LIN {X 0,Y 504.694,Z 139.15,A -85,B 0,C 180,E1 19601.04,E2 19601.04} C_VEL
LIN {X 0,Y 504.678,Z 139.182,A -85,B 0,C 180,E1 19597.642,E2 19597.642} C_VEL
LIN {X 0,Y 504.643,Z 139.158,A -85,B 0,C 180,E1 19594.284,E2 19594.284} C_VEL
LIN {X 0,Y 504.674,Z 139.176,A -85,B 0,C 180,E1 19590.889,E2 19590.889} C_VEL
LIN {X 0,Y 504.678,Z 139.173,A -85,B 0,C 180,E1 19587.527,E2 19587.527} C_VEL
LIN {X 0,Y 504.634,Z 139.159,A -85,B 0,C 180,E1 19584.13,E2 19584.13} C_VEL
LIN {X 0,Y 504.641,Z 139.168,A -85,B 0,C 180,E1 19580.597,E2 19580.597} C_VEL
LIN {X 0,Y 504.688,Z 139.169,A -85,B 0,C 180,E1 19577.193,E2 19577.193} C_VEL
LIN {X 0,Y 504.672,Z 139.48,A -85,B 0,C 180,E1 19576.287,E2 19576.287} C_VEL
LIN {X 0,Y 506.039,Z 142.777,A -85,B 0,C 180,E1 19575.775,E2 19575.775} C_VEL
LIN {X 0,Y 507.07,Z 144.526,A -85,B 0,C 180,E1 19575.494,E2 19575.494} C_VEL
LIN {X 0,Y 515.267,Z 161.516,A -85,B 0,C 180,E1 19573.08,E2 19573.08} C_VEL
LIN {X 0,Y 516.742,Z 164.473,A -85,B 0,C 180,E1 19572.673,E2 19572.673} C_VEL
LIN {X 0,Y 517.647,Z 168.38,A -85,B 0,C 180,E1 19572.251,E2 19572.251} C_VEL
LIN {X 0,Y 517.411,Z 174.74,A -85,B 0,C 180,E1 19571.749,E2 19571.749} C_VEL
LIN {X 0,Y 513.948,Z 193.541,A -85,B 0,C 180,E1 19570.561,E2 19570.561} C_VEL
LIN {X 0,Y 513.871,Z 194.507,A -85,B 0,C 180,E1 19570.49,E2 19570.49} C_VEL
LIN {X 0,Y 513.152,Z 207.74,A -85,B 0,C 180,E1 19569.537,E2 19569.537} C_VEL
LIN {X 0,Y 516.89,Z 230.706,A -85,B 0,C 180,E1 19568.755,E2 19568.755} C_VEL
LIN {X 0,Y 513.035,Z 451.518,A -85,B 0,C 180,E1 19565.211,E2 19565.211} C_VEL
LIN {X 0,Y 511.791,Z 516.033,A -85,B 0,C 180,E1 19564.149,E2 19564.149} C_VEL
LIN {X 0,Y 510.859,Z 536.785,A -85,B 0,C 180,E1 19563.612,E2 19563.612} C_VEL
LIN {X 0,Y 509.667,Z 559.479,A -85,B 0,C 180,E1 19562.815,E2 19562.815} C_VEL
LIN {X 0,Y 508.465,Z 579.082,A -85,B 0,C 180,E1 19561.935,E2 19561.935} C_VEL
LIN {X 0,Y 506.947,Z 599.576,A -85,B 0,C 180,E1 19560.784,E2 19560.784} C_VEL
LIN {X 0,Y 505.391,Z 619.262,A -85,B 0,C 180,E1 19559.447,E2 19559.447} C_VEL
LIN {X 0,Y 503.849,Z 637.518,A -85,B 0,C 180,E1 19557.984,E2 19557.984} C_VEL
LIN {X 0,Y 502.296,Z 655.386,A -85,B 0,C 180,E1 19556.288,E2 19556.288} C_VEL
LIN {X 0,Y 500.844,Z 671.992,A -85,B 0,C 180,E1 19554.448,E2 19554.448} C_VEL
LIN {X 0,Y 499.565,Z 687.373,A -85,B 0,C 180,E1 19552.474,E2 19552.474} C_VEL
LIN {X 0,Y 498.452,Z 701.856,A -85,B 0,C 180,E1 19550.305,E2 19550.305} C_VEL
LIN {X 0,Y 497.582,Z 714.282,A -85,B 0,C 180,E1 19548.109,E2 19548.109} C_VEL
LIN {X 0,Y 496.877,Z 726.123,A -85,B 0,C 180,E1 19545.643,E2 19545.643} C_VEL
LIN {X 0,Y 496.429,Z 735.604,A -85,B 0,C 180,E1 19543.274,E2 19543.274} C_VEL
LIN {X 0,Y 496.149,Z 743.247,A -85,B 0,C 180,E1 19540.919,E2 19540.919} C_VEL
LIN {X 0,Y 496,Z 749.548,A -85,B 0,C 180,E1 19538.462,E2 19538.462} C_VEL
LIN {X 0,Y 495.941,Z 754.255,A -85,B 0,C 180,E1 19536.018,E2 19536.018} C_VEL
LIN {X 0,Y 495.912,Z 757.243,A -85,B 0,C 180,E1 19533.583,E2 19533.583} C_VEL
LIN {X 0,Y 495.912,Z 758.793,A -85,B 0,C 180,E1 19531.04,E2 19531.04} C_VEL
LIN {X 0,Y 495.909,Z 758.744,A -85,B 0,C 180,E1 19528.614,E2 19528.614} C_VEL
LIN {X 0,Y 495.915,Z 757.105,A -85,B 0,C 180,E1 19526.185,E2 19526.185} C_VEL
LIN {X 0,Y 495.938,Z 753.899,A -85,B 0,C 180,E1 19523.688,E2 19523.688} C_VEL
LIN {X 0,Y 495.999,Z 749.235,A -85,B 0,C 180,E1 19521.304,E2 19521.304} C_VEL
LIN {X 0,Y 496.165,Z 742.811,A -85,B 0,C 180,E1 19518.846,E2 19518.846} C_VEL
LIN {X 0,Y 496.46,Z 735.096,A -85,B 0,C 180,E1 19516.49,E2 19516.49} C_VEL
LIN {X 0,Y 496.92,Z 725.442,A -85,B 0,C 180,E1 19514.11,E2 19514.11} C_VEL
LIN {X 0,Y 497.606,Z 713.924,A -85,B 0,C 180,E1 19511.733,E2 19511.733} C_VEL
LIN {X 0,Y 498.496,Z 701.2,A -85,B 0,C 180,E1 19509.502,E2 19509.502} C_VEL
LIN {X 0,Y 499.582,Z 687.135,A -85,B 0,C 180,E1 19507.402,E2 19507.402} C_VEL
LIN {X 0,Y 500.88,Z 671.569,A -85,B 0,C 180,E1 19505.411,E2 19505.411} C_VEL
LIN {X 0,Y 502.379,Z 654.427,A -85,B 0,C 180,E1 19503.525,E2 19503.525} C_VEL
LIN {X 0,Y 503.89,Z 637.058,A -85,B 0,C 180,E1 19501.884,E2 19501.884} C_VEL
LIN {X 0,Y 505.452,Z 618.551,A -85,B 0,C 180,E1 19500.41,E2 19500.41} C_VEL
LIN {X 0,Y 507.067,Z 597.939,A -85,B 0,C 180,E1 19499.027,E2 19499.027} C_VEL
LIN {X 0,Y 508.53,Z 578.192,A -85,B 0,C 180,E1 19497.933,E2 19497.933} C_VEL
LIN {X 0,Y 509.765,Z 557.764,A -85,B 0,C 180,E1 19497.025,E2 19497.025} C_VEL
LIN {X 0,Y 510.938,Z 535.278,A -85,B 0,C 180,E1 19496.253,E2 19496.253} C_VEL
LIN {X 0,Y 511.832,Z 514.323,A -85,B 0,C 180,E1 19495.728,E2 19495.728} C_VEL
LIN {X 0,Y 515.045,Z 335.958,A -85,B 0,C 180,E1 19492.843,E2 19492.843} C_VEL
LIN {X 0,Y 516.75,Z 228.784,A -85,B 0,C 180,E1 19491.107,E2 19491.107} C_VEL
LIN {X 0,Y 513.075,Z 206.394,A -85,B 0,C 180,E1 19490.302,E2 19490.302} C_VEL
LIN {X 0,Y 514.845,Z 178.717,A -85,B 0,C 180,E1 19488.224,E2 19488.224} C_VEL
LIN {X 0,Y 506.945,Z 161.195,A -85,B 0,C 180,E1 19485.876,E2 19485.876} C_VEL
LIN {X 0,Y 500.724,Z 148.664,A -85,B 0,C 180,E1 19484.019,E2 19484.019} C_VEL
LIN {X 0,Y 498.026,Z 143.652,A -85,B 0,C 180,E1 19483.218,E2 19483.218} C_VEL
LIN {X 0,Y 496.796,Z 140.454,A -85,B 0,C 180,E1 19482.707,E2 19482.707} C_VEL
LIN {X 0,Y 496.708,Z 140.147,A -85,B 0,C 180,E1 19480.253,E2 19480.253} C_VEL
LIN {X 0,Y 496.74,Z 140.151,A -85,B 0,C 180,E1 19476.858,E2 19476.858} C_VEL
LIN {X 0,Y 496.699,Z 140.176,A -85,B 0,C 180,E1 19473.475,E2 19473.475} C_VEL
LIN {X 0,Y 496.698,Z 140.155,A -85,B 0,C 180,E1 19469.949,E2 19469.949} C_VEL
LIN {X 0,Y 496.757,Z 140.151,A -85,B 0,C 180,E1 19466.665,E2 19466.665} C_VEL
LIN {X 0,Y 496.721,Z 140.167,A -85,B 0,C 180,E1 19463.237,E2 19463.237} C_VEL
LIN {X 0,Y 496.706,Z 140.144,A -85,B 0,C 180,E1 19459.766,E2 19459.766} C_VEL
LIN {X 0,Y 496.742,Z 140.172,A -85,B 0,C 180,E1 19456.368,E2 19456.368} C_VEL
LIN {X 0,Y 496.76,Z 140.17,A -85,B 0,C 180,E1 19452.91,E2 19452.91} C_VEL
LIN {X 0,Y 496.722,Z 140.171,A -85,B 0,C 180,E1 19449.496,E2 19449.496} C_VEL
LIN {X 0,Y 496.723,Z 140.171,A -85,B 0,C 180,E1 19445.892,E2 19445.892} C_VEL
LIN {X 0,Y 496.758,Z 140.169,A -85,B 0,C 180,E1 19442.423,E2 19442.423} C_VEL
LIN {X 0,Y 496.766,Z 140.168,A -85,B 0,C 180,E1 19438.962,E2 19438.962} C_VEL
LIN {X 0,Y 496.733,Z 140.168,A -85,B 0,C 180,E1 19435.498,E2 19435.498} C_VEL
LIN {X 0,Y 496.734,Z 140.168,A -85,B 0,C 180,E1 19431.9,E2 19431.9} C_VEL
LIN {X 0,Y 496.763,Z 140.166,A -85,B 0,C 180,E1 19428.389,E2 19428.389} C_VEL
LIN {X 0,Y 496.768,Z 140.132,A -85,B 0,C 180,E1 19424.832,E2 19424.832} C_VEL
LIN {X 0,Y 496.753,Z 140.172,A -85,B 0,C 180,E1 19421.335,E2 19421.335} C_VEL
LIN {X 0,Y 496.74,Z 140.141,A -85,B 0,C 180,E1 19417.765,E2 19417.765} C_VEL
LIN {X 0,Y 496.761,Z 140.16,A -85,B 0,C 180,E1 19414.23,E2 19414.23} C_VEL
LIN {X 0,Y 496.768,Z 140.169,A -85,B 0,C 180,E1 19410.632,E2 19410.632} C_VEL
LIN {X 0,Y 496.765,Z 140.142,A -85,B 0,C 180,E1 19407.065,E2 19407.065} C_VEL
LIN {X 0,Y 496.752,Z 140.144,A -85,B 0,C 180,E1 19403.575,E2 19403.575} C_VEL
LIN {X 0,Y 496.76,Z 140.147,A -85,B 0,C 180,E1 19400.054,E2 19400.054} C_VEL
LIN {X 0,Y 496.807,Z 140.5,A -85,B 0,C 180,E1 19399.563,E2 19399.563} C_VEL
LIN {X 0,Y 498.398,Z 144.079,A -85,B 0,C 180,E1 19399.004,E2 19399.004} C_VEL
LIN {X 0,Y 499.562,Z 146.324,A -85,B 0,C 180,E1 19398.663,E2 19398.663} C_VEL
LIN {X 0,Y 505.939,Z 158.646,A -85,B 0,C 180,E1 19396.861,E2 19396.861} C_VEL
LIN {X 0,Y 509.151,Z 164.9,A -85,B 0,C 180,E1 19396.037,E2 19396.037} C_VEL
LIN {X 0,Y 521.412,Z 183.553,A -85,B 0,C 180,E1 19394.429,E2 19394.429} C_VEL
LIN {X 0,Y 521.63,Z 187.591,A -85,B 0,C 180,E1 19394.333,E2 19394.333} C_VEL
LIN {X 0,Y 518.314,Z 393.262,A -85,B 0,C 180,E1 19390.993,E2 19390.993} C_VEL
LIN {X 0,Y 516.548,Z 508.593,A -85,B 0,C 180,E1 19389.158,E2 19389.158} C_VEL
LIN {X 0,Y 515.582,Z 532.711,A -85,B 0,C 180,E1 19388.591,E2 19388.591} C_VEL
LIN {X 0,Y 514.484,Z 552.35,A -85,B 0,C 180,E1 19387.957,E2 19387.957} C_VEL
LIN {X 0,Y 512.962,Z 574.834,A -85,B 0,C 180,E1 19387.033,E2 19387.033} C_VEL
LIN {X 0,Y 511.337,Z 595.456,A -85,B 0,C 180,E1 19385.978,E2 19385.978} C_VEL
LIN {X 0,Y 509.442,Z 617.344,A -85,B 0,C 180,E1 19384.623,E2 19384.623} C_VEL
LIN {X 0,Y 507.601,Z 636.829,A -85,B 0,C 180,E1 19383.201,E2 19383.201} C_VEL
LIN {X 0,Y 505.71,Z 656.021,A -85,B 0,C 180,E1 19381.554,E2 19381.554} C_VEL
LIN {X 0,Y 503.886,Z 674.456,A -85,B 0,C 180,E1 19379.74,E2 19379.74} C_VEL
LIN {X 0,Y 502.167,Z 691.624,A -85,B 0,C 180,E1 19377.769,E2 19377.769} C_VEL
LIN {X 0,Y 500.564,Z 708.453,A -85,B 0,C 180,E1 19375.559,E2 19375.559} C_VEL
LIN {X 0,Y 499.286,Z 722.975,A -85,B 0,C 180,E1 19373.359,E2 19373.359} C_VEL
LIN {X 0,Y 498.176,Z 736.82,A -85,B 0,C 180,E1 19370.931,E2 19370.931} C_VEL
LIN {X 0,Y 497.355,Z 748.726,A -85,B 0,C 180,E1 19368.519,E2 19368.519} C_VEL
LIN {X 0,Y 496.736,Z 759.152,A -85,B 0,C 180,E1 19366.007,E2 19366.007} C_VEL
LIN {X 0,Y 496.335,Z 768.425,A -85,B 0,C 180,E1 19363.347,E2 19363.347} C_VEL
LIN {X 0,Y 496.104,Z 775.261,A -85,B 0,C 180,E1 19360.92,E2 19360.92} C_VEL
LIN {X 0,Y 495.975,Z 781.308,A -85,B 0,C 180,E1 19358.18,E2 19358.18} C_VEL
LIN {X 0,Y 495.918,Z 785.119,A -85,B 0,C 180,E1 19355.786,E2 19355.786} C_VEL
LIN {X 0,Y 495.911,Z 787.85,A -85,B 0,C 180,E1 19353.12,E2 19353.12} C_VEL
LIN {X 0,Y 495.901,Z 788.872,A -85,B 0,C 180,E1 19350.693,E2 19350.693} C_VEL
LIN {X 0,Y 495.907,Z 788.526,A -85,B 0,C 180,E1 19348.036,E2 19348.036} C_VEL
LIN {X 0,Y 495.903,Z 786.729,A -85,B 0,C 180,E1 19345.606,E2 19345.606} C_VEL
LIN {X 0,Y 495.948,Z 783.494,A -85,B 0,C 180,E1 19343.052,E2 19343.052} C_VEL
LIN {X 0,Y 496.015,Z 778.574,A -85,B 0,C 180,E1 19340.486,E2 19340.486} C_VEL
LIN {X 0,Y 496.199,Z 772.175,A -85,B 0,C 180,E1 19337.904,E2 19337.904} C_VEL
LIN {X 0,Y 496.494,Z 764.344,A -85,B 0,C 180,E1 19335.421,E2 19335.421} C_VEL
LIN {X 0,Y 497.004,Z 754.423,A -85,B 0,C 180,E1 19332.799,E2 19332.799} C_VEL
LIN {X 0,Y 497.694,Z 743.578,A -85,B 0,C 180,E1 19330.398,E2 19330.398} C_VEL
LIN {X 0,Y 498.691,Z 730.158,A -85,B 0,C 180,E1 19327.857,E2 19327.857} C_VEL
LIN {X 0,Y 499.892,Z 716.017,A -85,B 0,C 180,E1 19325.542,E2 19325.542} C_VEL
LIN {X 0,Y 501.341,Z 700.156,A -85,B 0,C 180,E1 19323.313,E2 19323.313} C_VEL
LIN {X 0,Y 503.003,Z 683.24,A -85,B 0,C 180,E1 19321.236,E2 19321.236} C_VEL
LIN {X 0,Y 504.71,Z 665.965,A -85,B 0,C 180,E1 19319.395,E2 19319.395} C_VEL
LIN {X 0,Y 506.661,Z 646.455,A -85,B 0,C 180,E1 19317.597,E2 19317.597} C_VEL
LIN {X 0,Y 508.468,Z 627.905,A -85,B 0,C 180,E1 19316.119,E2 19316.119} C_VEL
LIN {X 0,Y 510.36,Z 606.838,A -85,B 0,C 180,E1 19314.695,E2 19314.695} C_VEL
LIN {X 0,Y 512.133,Z 586.304,A -85,B 0,C 180,E1 19313.525,E2 19313.525} C_VEL
LIN {X 0,Y 513.647,Z 565.101,A -85,B 0,C 180,E1 19312.541,E2 19312.541} C_VEL
LIN {X 0,Y 515.036,Z 543.176,A -85,B 0,C 180,E1 19311.718,E2 19311.718} C_VEL
LIN {X 0,Y 516.102,Z 520.863,A -85,B 0,C 180,E1 19311.103,E2 19311.103} C_VEL
LIN {X 0,Y 516.876,Z 496.406,A -85,B 0,C 180,E1 19310.628,E2 19310.628} C_VEL
LIN {X 0,Y 519.924,Z 286.714,A -85,B 0,C 180,E1 19307.299,E2 19307.299} C_VEL
LIN {X 0,Y 521.507,Z 184.101,A -85,B 0,C 180,E1 19305.591,E2 19305.591} C_VEL
LIN {X 0,Y 520.746,Z 182.337,A -85,B 0,C 180,E1 19305.484,E2 19305.484} C_VEL
LIN {X 0,Y 508.362,Z 163.559,A -85,B 0,C 180,E1 19303.814,E2 19303.814} C_VEL
LIN {X 0,Y 500.755,Z 148.542,A -85,B 0,C 180,E1 19301.674,E2 19301.674} C_VEL
LIN {X 0,Y 498.393,Z 144.075,A -85,B 0,C 180,E1 19300.996,E2 19300.996} C_VEL
LIN {X 0,Y 496.81,Z 140.516,A -85,B 0,C 180,E1 19300.437,E2 19300.437} C_VEL
LIN {X 0,Y 496.769,Z 140.15,A -85,B 0,C 180,E1 19299.75,E2 19299.75} C_VEL
LIN {X 0,Y 496.751,Z 140.147,A -85,B 0,C 180,E1 19296.186,E2 19296.186} C_VEL
LIN {X 0,Y 496.759,Z 140.141,A -85,B 0,C 180,E1 19292.644,E2 19292.644} C_VEL
LIN {X 0,Y 496.765,Z 140.163,A -85,B 0,C 180,E1 19289.132,E2 19289.132} C_VEL
LIN {X 0,Y 496.768,Z 140.16,A -85,B 0,C 180,E1 19285.513,E2 19285.513} C_VEL
LIN {X 0,Y 496.744,Z 140.138,A -85,B 0,C 180,E1 19281.986,E2 19281.986} C_VEL
LIN {X 0,Y 496.744,Z 140.17,A -85,B 0,C 180,E1 19278.422,E2 19278.422} C_VEL
LIN {X 0,Y 496.768,Z 140.134,A -85,B 0,C 180,E1 19274.929,E2 19274.929} C_VEL
LIN {X 0,Y 496.77,Z 140.167,A -85,B 0,C 180,E1 19271.376,E2 19271.376} C_VEL
LIN {X 0,Y 496.746,Z 140.166,A -85,B 0,C 180,E1 19267.867,E2 19267.867} C_VEL
LIN {X 0,Y 496.733,Z 140.167,A -85,B 0,C 180,E1 19264.387,E2 19264.387} C_VEL
LIN {X 0,Y 496.761,Z 140.167,A -85,B 0,C 180,E1 19260.922,E2 19260.922} C_VEL
LIN {X 0,Y 496.77,Z 140.17,A -85,B 0,C 180,E1 19257.347,E2 19257.347} C_VEL
LIN {X 0,Y 496.735,Z 140.17,A -85,B 0,C 180,E1 19253.876,E2 19253.876} C_VEL
LIN {X 0,Y 496.723,Z 140.17,A -85,B 0,C 180,E1 19250.382,E2 19250.382} C_VEL
LIN {X 0,Y 496.754,Z 140.169,A -85,B 0,C 180,E1 19246.947,E2 19246.947} C_VEL
LIN {X 0,Y 496.756,Z 140.171,A -85,B 0,C 180,E1 19243.513,E2 19243.513} C_VEL
LIN {X 0,Y 496.712,Z 140.145,A -85,B 0,C 180,E1 19240.055,E2 19240.055} C_VEL
LIN {X 0,Y 496.714,Z 140.166,A -85,B 0,C 180,E1 19236.511,E2 19236.511} C_VEL
LIN {X 0,Y 496.755,Z 140.155,A -85,B 0,C 180,E1 19233.072,E2 19233.072} C_VEL
LIN {X 0,Y 496.728,Z 140.147,A -85,B 0,C 180,E1 19229.653,E2 19229.653} C_VEL
LIN {X 0,Y 496.7,Z 140.176,A -85,B 0,C 180,E1 19226.237,E2 19226.237} C_VEL
LIN {X 0,Y 496.711,Z 140.164,A -85,B 0,C 180,E1 19222.706,E2 19222.706} C_VEL
LIN {X 0,Y 496.75,Z 140.143,A -85,B 0,C 180,E1 19219.359,E2 19219.359} C_VEL
LIN {X 0,Y 496.78,Z 140.382,A -85,B 0,C 180,E1 19217.22,E2 19217.22} C_VEL
LIN {X 0,Y 498.164,Z 143.861,A -85,B 0,C 180,E1 19216.652,E2 19216.652} C_VEL
LIN {X 0,Y 499.353,Z 146.181,A -85,B 0,C 180,E1 19216.287,E2 19216.287} C_VEL
LIN {X 0,Y 503.375,Z 154.077,A -85,B 0,C 180,E1 19215.079,E2 19215.079} C_VEL
LIN {X 0,Y 511.075,Z 170.103,A -85,B 0,C 180,E1 19212.807,E2 19212.807} C_VEL
LIN {X 0,Y 514.903,Z 179.032,A -85,B 0,C 180,E1 19211.654,E2 19211.654} C_VEL
LIN {X 0,Y 513.871,Z 194.507,A -85,B 0,C 180,E1 19210.49,E2 19210.49} C_VEL
LIN {X 0,Y 512.881,Z 199.17,A -85,B 0,C 180,E1 19210.24,E2 19210.24} C_VEL
LIN {X 0,Y 509.36,Z 209.118,A -85,B 0,C 180,E1 19210.022,E2 19210.022} C_VEL
LIN {X 0,Y 508.39,Z 215.006,A -85,B 0,C 180,E1 19209.904,E2 19209.904} C_VEL
LIN {X 0,Y 508.565,Z 217.173,A -85,B 0,C 180,E1 19209.836,E2 19209.836} C_VEL
LIN {X 0,Y 510.869,Z 232.395,A -85,B 0,C 180,E1 19209.324,E2 19209.324} C_VEL
LIN {X 0,Y 506.778,Z 455.91,A -85,B 0,C 180,E1 19205.716,E2 19205.716} C_VEL
LIN {X 0,Y 505.532,Z 516.179,A -85,B 0,C 180,E1 19204.714,E2 19204.714} C_VEL
LIN {X 0,Y 504.544,Z 536.826,A -85,B 0,C 180,E1 19204.176,E2 19204.176} C_VEL
LIN {X 0,Y 503.294,Z 557.406,A -85,B 0,C 180,E1 19203.448,E2 19203.448} C_VEL
LIN {X 0,Y 501.851,Z 577.174,A -85,B 0,C 180,E1 19202.542,E2 19202.542} C_VEL
LIN {X 0,Y 499.97,Z 599.586,A -85,B 0,C 180,E1 19201.261,E2 19201.261} C_VEL
LIN {X 0,Y 498.281,Z 619.335,A -85,B 0,C 180,E1 19199.904,E2 19199.904} C_VEL
LIN {X 0,Y 496.623,Z 637.47,A -85,B 0,C 180,E1 19198.433,E2 19198.433} C_VEL
LIN {X 0,Y 494.936,Z 655.331,A -85,B 0,C 180,E1 19196.717,E2 19196.717} C_VEL
LIN {X 0,Y 493.36,Z 671.816,A -85,B 0,C 180,E1 19194.867,E2 19194.867} C_VEL
LIN {X 0,Y 491.95,Z 687.379,A -85,B 0,C 180,E1 19192.842,E2 19192.842} C_VEL
LIN {X 0,Y 490.726,Z 701.86,A -85,B 0,C 180,E1 19190.639,E2 19190.639} C_VEL
LIN {X 0,Y 489.781,Z 714.088,A -85,B 0,C 180,E1 19188.446,E2 19188.446} C_VEL
LIN {X 0,Y 489.025,Z 725.61,A -85,B 0,C 180,E1 19186.022,E2 19186.022} C_VEL
LIN {X 0,Y 488.518,Z 735.2,A -85,B 0,C 180,E1 19183.613,E2 19183.613} C_VEL
LIN {X 0,Y 488.188,Z 743.028,A -85,B 0,C 180,E1 19181.174,E2 19181.174} C_VEL
LIN {X 0,Y 488.007,Z 749.55,A -85,B 0,C 180,E1 19178.602,E2 19178.602} C_VEL
LIN {X 0,Y 487.943,Z 754.256,A -85,B 0,C 180,E1 19176.117,E2 19176.117} C_VEL
LIN {X 0,Y 487.912,Z 757.254,A -85,B 0,C 180,E1 19173.632,E2 19173.632} C_VEL
LIN {X 0,Y 487.911,Z 758.793,A -85,B 0,C 180,E1 19171.057,E2 19171.057} C_VEL
LIN {X 0,Y 487.909,Z 758.744,A -85,B 0,C 180,E1 19168.591,E2 19168.591} C_VEL
LIN {X 0,Y 487.915,Z 757.104,A -85,B 0,C 180,E1 19166.123,E2 19166.123} C_VEL
LIN {X 0,Y 487.94,Z 753.987,A -85,B 0,C 180,E1 19163.635,E2 19163.635} C_VEL
LIN {X 0,Y 488.006,Z 749.488,A -85,B 0,C 180,E1 19161.28,E2 19161.28} C_VEL
LIN {X 0,Y 488.2,Z 742.808,A -85,B 0,C 180,E1 19158.661,E2 19158.661} C_VEL
LIN {X 0,Y 488.525,Z 735.094,A -85,B 0,C 180,E1 19156.266,E2 19156.266} C_VEL
LIN {X 0,Y 489.033,Z 725.475,A -85,B 0,C 180,E1 19153.856,E2 19153.856} C_VEL
LIN {X 0,Y 489.793,Z 713.918,A -85,B 0,C 180,E1 19151.431,E2 19151.431} C_VEL
LIN {X 0,Y 490.743,Z 701.647,A -85,B 0,C 180,E1 19149.237,E2 19149.237} C_VEL
LIN {X 0,Y 491.971,Z 687.13,A -85,B 0,C 180,E1 19147.033,E2 19147.033} C_VEL
LIN {X 0,Y 493.388,Z 671.516,A -85,B 0,C 180,E1 19145.006,E2 19145.006} C_VEL
LIN {X 0,Y 495.019,Z 654.417,A -85,B 0,C 180,E1 19143.1,E2 19143.1} C_VEL
LIN {X 0,Y 496.668,Z 637.048,A -85,B 0,C 180,E1 19141.438,E2 19141.438} C_VEL
LIN {X 0,Y 498.334,Z 618.748,A -85,B 0,C 180,E1 19139.961,E2 19139.961} C_VEL
LIN {X 0,Y 500.023,Z 598.93,A -85,B 0,C 180,E1 19138.608,E2 19138.608} C_VEL
LIN {X 0,Y 501.83,Z 577.591,A -85,B 0,C 180,E1 19137.389,E2 19137.389} C_VEL
LIN {X 0,Y 503.274,Z 557.725,A -85,B 0,C 180,E1 19136.476,E2 19136.476} C_VEL
LIN {X 0,Y 504.561,Z 536.539,A -85,B 0,C 180,E1 19135.725,E2 19135.725} C_VEL
LIN {X 0,Y 505.546,Z 515.794,A -85,B 0,C 180,E1 19135.188,E2 19135.188} C_VEL
LIN {X 0,Y 507.26,Z 430.463,A -85,B 0,C 180,E1 19133.783,E2 19133.783} C_VEL
LIN {X 0,Y 510.875,Z 231.206,A -85,B 0,C 180,E1 19130.565,E2 19130.565} C_VEL
LIN {X 0,Y 506.744,Z 206.374,A -85,B 0,C 180,E1 19129.672,E2 19129.672} C_VEL
LIN {X 0,Y 508.341,Z 182.535,A -85,B 0,C 180,E1 19127.862,E2 19127.862} C_VEL
LIN {X 0,Y 500.93,Z 166.019,A -85,B 0,C 180,E1 19125.608,E2 19125.608} C_VEL
LIN {X 0,Y 494.73,Z 153.561,A -85,B 0,C 180,E1 19123.724,E2 19123.724} C_VEL
LIN {X 0,Y 490.638,Z 145.354,A -85,B 0,C 180,E1 19122.418,E2 19122.418} C_VEL
LIN {X 0,Y 488.884,Z 141.905,A -85,B 0,C 180,E1 19121.841,E2 19121.841} C_VEL
LIN {X 0,Y 488.756,Z 141.162,A -85,B 0,C 180,E1 19121.521,E2 19121.521} C_VEL
LIN {X 0,Y 488.752,Z 141.168,A -85,B 0,C 180,E1 19117.859,E2 19117.859} C_VEL
LIN {X 0,Y 488.785,Z 141.147,A -85,B 0,C 180,E1 19114.374,E2 19114.374} C_VEL
LIN {X 0,Y 488.804,Z 141.128,A -85,B 0,C 180,E1 19110.892,E2 19110.892} C_VEL
LIN {X 0,Y 488.764,Z 141.165,A -85,B 0,C 180,E1 19107.537,E2 19107.537} C_VEL
LIN {X 0,Y 488.766,Z 141.149,A -85,B 0,C 180,E1 19103.88,E2 19103.88} C_VEL
LIN {X 0,Y 488.808,Z 141.137,A -85,B 0,C 180,E1 19100.474,E2 19100.474} C_VEL
LIN {X 0,Y 488.818,Z 141.151,A -85,B 0,C 180,E1 19096.885,E2 19096.885} C_VEL
LIN {X 0,Y 488.781,Z 141.156,A -85,B 0,C 180,E1 19093.486,E2 19093.486} C_VEL
LIN {X 0,Y 488.781,Z 141.159,A -85,B 0,C 180,E1 19089.895,E2 19089.895} C_VEL
LIN {X 0,Y 488.82,Z 141.157,A -85,B 0,C 180,E1 19086.46,E2 19086.46} C_VEL
LIN {X 0,Y 488.823,Z 141.153,A -85,B 0,C 180,E1 19082.931,E2 19082.931} C_VEL
LIN {X 0,Y 488.795,Z 141.154,A -85,B 0,C 180,E1 19079.414,E2 19079.414} C_VEL
LIN {X 0,Y 488.792,Z 141.155,A -85,B 0,C 180,E1 19075.895,E2 19075.895} C_VEL
LIN {X 0,Y 488.823,Z 141.154,A -85,B 0,C 180,E1 19072.36,E2 19072.36} C_VEL
LIN {X 0,Y 488.831,Z 141.153,A -85,B 0,C 180,E1 19068.796,E2 19068.796} C_VEL
LIN {X 0,Y 488.816,Z 141.123,A -85,B 0,C 180,E1 19065.186,E2 19065.186} C_VEL
LIN {X 0,Y 488.803,Z 141.159,A -85,B 0,C 180,E1 19061.639,E2 19061.639} C_VEL
LIN {X 0,Y 488.806,Z 141.124,A -85,B 0,C 180,E1 19058.017,E2 19058.017} C_VEL
LIN {X 0,Y 488.83,Z 141.149,A -85,B 0,C 180,E1 19054.562,E2 19054.562} C_VEL
LIN {X 0,Y 488.829,Z 141.147,A -85,B 0,C 180,E1 19051.003,E2 19051.003} C_VEL
LIN {X 0,Y 488.815,Z 141.128,A -85,B 0,C 180,E1 19047.428,E2 19047.428} C_VEL
LIN {X 0,Y 488.813,Z 141.134,A -85,B 0,C 180,E1 19043.895,E2 19043.895} C_VEL
LIN {X 0,Y 488.848,Z 141.33,A -85,B 0,C 180,E1 19040.582,E2 19040.582} C_VEL
LIN {X 0,Y 489.41,Z 143.288,A -85,B 0,C 180,E1 19040.249,E2 19040.249} C_VEL
LIN {X 0,Y 491.407,Z 146.632,A -85,B 0,C 180,E1 19039.682,E2 19039.682} C_VEL
LIN {X 0,Y 500,Z 163.323,A -85,B 0,C 180,E1 19037.164,E2 19037.164} C_VEL
LIN {X 0,Y 501.695,Z 166.359,A -85,B 0,C 180,E1 19036.817,E2 19036.817} C_VEL
LIN {X 0,Y 515.665,Z 187.341,A -85,B 0,C 180,E1 19034.931,E2 19034.931} C_VEL
LIN {X 0,Y 512.047,Z 386.592,A -85,B 0,C 180,E1 19031.642,E2 19031.642} C_VEL
LIN {X 0,Y 509.974,Z 511.991,A -85,B 0,C 180,E1 19029.62,E2 19029.62} C_VEL
LIN {X 0,Y 509.01,Z 534.811,A -85,B 0,C 180,E1 19029.066,E2 19029.066} C_VEL
LIN {X 0,Y 507.865,Z 556.069,A -85,B 0,C 180,E1 19028.377,E2 19028.377} C_VEL
LIN {X 0,Y 506.275,Z 577.4,A -85,B 0,C 180,E1 19027.464,E2 19027.464} C_VEL
LIN {X 0,Y 504.494,Z 598.725,A -85,B 0,C 180,E1 19026.34,E2 19026.34} C_VEL
LIN {X 0,Y 502.521,Z 619.141,A -85,B 0,C 180,E1 19025.03,E2 19025.03} C_VEL
LIN {X 0,Y 500.474,Z 639.187,A -85,B 0,C 180,E1 19023.531,E2 19023.531} C_VEL
LIN {X 0,Y 498.423,Z 658.271,A -85,B 0,C 180,E1 19021.842,E2 19021.842} C_VEL
LIN {X 0,Y 496.283,Z 677.792,A -85,B 0,C 180,E1 19019.842,E2 19019.842} C_VEL
LIN {X 0,Y 494.577,Z 693.896,A -85,B 0,C 180,E1 19017.938,E2 19017.938} C_VEL
LIN {X 0,Y 492.878,Z 710.145,A -85,B 0,C 180,E1 19015.729,E2 19015.729} C_VEL
LIN {X 0,Y 491.448,Z 725.23,A -85,B 0,C 180,E1 19013.373,E2 19013.373} C_VEL
LIN {X 0,Y 490.322,Z 738.088,A -85,B 0,C 180,E1 19011.032,E2 19011.032} C_VEL
LIN {X 0,Y 489.409,Z 750.291,A -85,B 0,C 180,E1 19008.461,E2 19008.461} C_VEL
LIN {X 0,Y 488.784,Z 760.069,A -85,B 0,C 180,E1 19006.03,E2 19006.03} C_VEL
LIN {X 0,Y 488.341,Z 769.35,A -85,B 0,C 180,E1 19003.256,E2 19003.256} C_VEL
LIN {X 0,Y 488.104,Z 776.169,A -85,B 0,C 180,E1 19000.743,E2 19000.743} C_VEL
LIN {X 0,Y 487.976,Z 781.842,A -85,B 0,C 180,E1 18998.009,E2 18998.009} C_VEL
LIN {X 0,Y 487.915,Z 785.437,A -85,B 0,C 180,E1 18995.645,E2 18995.645} C_VEL
LIN {X 0,Y 487.914,Z 787.986,A -85,B 0,C 180,E1 18992.937,E2 18992.937} C_VEL
LIN {X 0,Y 487.899,Z 788.895,A -85,B 0,C 180,E1 18990.587,E2 18990.587} C_VEL
LIN {X 0,Y 487.907,Z 788.459,A -85,B 0,C 180,E1 18987.886,E2 18987.886} C_VEL
LIN {X 0,Y 487.903,Z 786.729,A -85,B 0,C 180,E1 18985.534,E2 18985.534} C_VEL
LIN {X 0,Y 487.954,Z 783.494,A -85,B 0,C 180,E1 18982.938,E2 18982.938} C_VEL
LIN {X 0,Y 488.025,Z 778.574,A -85,B 0,C 180,E1 18980.329,E2 18980.329} C_VEL
LIN {X 0,Y 488.235,Z 772.174,A -85,B 0,C 180,E1 18977.703,E2 18977.703} C_VEL
LIN {X 0,Y 488.564,Z 764.343,A -85,B 0,C 180,E1 18975.179,E2 18975.179} C_VEL
LIN {X 0,Y 489.127,Z 754.421,A -85,B 0,C 180,E1 18972.513,E2 18972.513} C_VEL
LIN {X 0,Y 489.89,Z 743.58,A -85,B 0,C 180,E1 18970.072,E2 18970.072} C_VEL
LIN {X 0,Y 490.993,Z 730.156,A -85,B 0,C 180,E1 18967.491,E2 18967.491} C_VEL
LIN {X 0,Y 492.316,Z 716.019,A -85,B 0,C 180,E1 18965.141,E2 18965.141} C_VEL
LIN {X 0,Y 493.876,Z 700.339,A -85,B 0,C 180,E1 18962.903,E2 18962.903} C_VEL
LIN {X 0,Y 495.763,Z 682.786,A -85,B 0,C 180,E1 18960.721,E2 18960.721} C_VEL
LIN {X 0,Y 497.62,Z 665.545,A -85,B 0,C 180,E1 18958.865,E2 18958.865} C_VEL
LIN {X 0,Y 499.764,Z 645.793,A -85,B 0,C 180,E1 18957.032,E2 18957.032} C_VEL
LIN {X 0,Y 501.818,Z 626.28,A -85,B 0,C 180,E1 18955.47,E2 18955.47} C_VEL
LIN {X 0,Y 503.805,Z 605.828,A -85,B 0,C 180,E1 18954.095,E2 18954.095} C_VEL
LIN {X 0,Y 505.707,Z 585.104,A -85,B 0,C 180,E1 18952.914,E2 18952.914} C_VEL
LIN {X 0,Y 507.284,Z 564.192,A -85,B 0,C 180,E1 18951.945,E2 18951.945} C_VEL
LIN {X 0,Y 508.622,Z 542.702,A -85,B 0,C 180,E1 18951.161,E2 18951.161} C_VEL
LIN {X 0,Y 509.64,Z 520.432,A -85,B 0,C 180,E1 18950.565,E2 18950.565} C_VEL
LIN {X 0,Y 510.377,Z 494.754,A -85,B 0,C 180,E1 18950.082,E2 18950.082} C_VEL
LIN {X 0,Y 513.684,Z 290.898,A -85,B 0,C 180,E1 18946.797,E2 18946.797} C_VEL
LIN {X 0,Y 515.488,Z 187.094,A -85,B 0,C 180,E1 18945.05,E2 18945.05} C_VEL
LIN {X 0,Y 500.594,Z 164.637,A -85,B 0,C 180,E1 18943.007,E2 18943.007} C_VEL
LIN {X 0,Y 493.349,Z 150.221,A -85,B 0,C 180,E1 18940.89,E2 18940.89} C_VEL
LIN {X 0,Y 491.232,Z 146.083,A -85,B 0,C 180,E1 18940.248,E2 18940.248} C_VEL
LIN {X 0,Y 489.091,Z 142.404,A -85,B 0,C 180,E1 18939.63,E2 18939.63} C_VEL
LIN {X 0,Y 488.83,Z 141.205,A -85,B 0,C 180,E1 18939.351,E2 18939.351} C_VEL
LIN {X 0,Y 488.828,Z 141.139,A -85,B 0,C 180,E1 18935.707,E2 18935.707} C_VEL
LIN {X 0,Y 488.81,Z 141.129,A -85,B 0,C 180,E1 18932.129,E2 18932.129} C_VEL
LIN {X 0,Y 488.818,Z 141.142,A -85,B 0,C 180,E1 18928.596,E2 18928.596} C_VEL
LIN {X 0,Y 488.83,Z 141.154,A -85,B 0,C 180,E1 18925.029,E2 18925.029} C_VEL
LIN {X 0,Y 488.829,Z 141.12,A -85,B 0,C 180,E1 18921.465,E2 18921.465} C_VEL
LIN {X 0,Y 488.814,Z 141.156,A -85,B 0,C 180,E1 18917.868,E2 18917.868} C_VEL
LIN {X 0,Y 488.797,Z 141.131,A -85,B 0,C 180,E1 18914.33,E2 18914.33} C_VEL
LIN {X 0,Y 488.819,Z 141.15,A -85,B 0,C 180,E1 18910.847,E2 18910.847} C_VEL
LIN {X 0,Y 488.834,Z 141.15,A -85,B 0,C 180,E1 18907.257,E2 18907.257} C_VEL
LIN {X 0,Y 488.818,Z 141.151,A -85,B 0,C 180,E1 18903.635,E2 18903.635} C_VEL
LIN {X 0,Y 488.789,Z 141.152,A -85,B 0,C 180,E1 18900.117,E2 18900.117} C_VEL
LIN {X 0,Y 488.79,Z 141.151,A -85,B 0,C 180,E1 18896.482,E2 18896.482} C_VEL
LIN {X 0,Y 488.818,Z 141.151,A -85,B 0,C 180,E1 18892.95,E2 18892.95} C_VEL
LIN {X 0,Y 488.826,Z 141.151,A -85,B 0,C 180,E1 18889.392,E2 18889.392} C_VEL
LIN {X 0,Y 488.787,Z 141.154,A -85,B 0,C 180,E1 18885.911,E2 18885.911} C_VEL
LIN {X 0,Y 488.775,Z 141.149,A -85,B 0,C 180,E1 18882.377,E2 18882.377} C_VEL
LIN {X 0,Y 488.8,Z 141.148,A -85,B 0,C 180,E1 18878.866,E2 18878.866} C_VEL
LIN {X 0,Y 488.81,Z 141.131,A -85,B 0,C 180,E1 18875.466,E2 18875.466} C_VEL
LIN {X 0,Y 488.77,Z 141.163,A -85,B 0,C 180,E1 18872.066,E2 18872.066} C_VEL
LIN {X 0,Y 488.763,Z 141.137,A -85,B 0,C 180,E1 18868.419,E2 18868.419} C_VEL
LIN {X 0,Y 488.802,Z 141.135,A -85,B 0,C 180,E1 18865.058,E2 18865.058} C_VEL
LIN {X 0,Y 488.792,Z 141.159,A -85,B 0,C 180,E1 18861.548,E2 18861.548} C_VEL
LIN {X 0,Y 488.765,Z 141.247,A -85,B 0,C 180,E1 18858.251,E2 18858.251} C_VEL
LIN {X 0,Y 489.066,Z 142.574,A -85,B 0,C 180,E1 18857.968,E2 18857.968} C_VEL
LIN {X 0,Y 491.287,Z 146.623,A -85,B 0,C 180,E1 18857.28,E2 18857.28} C_VEL
LIN {X 0,Y 497.95,Z 160.078,A -85,B 0,C 180,E1 18855.187,E2 18855.187} C_VEL
LIN {X 0,Y 505.214,Z 175.257,A -85,B 0,C 180,E1 18853.007,E2 18853.007} C_VEL
LIN {X 0,Y 508.424,Z 182.735,A -85,B 0,C 180,E1 18852.023,E2 18852.023} C_VEL
LIN {X 0,Y 506.821,Z 207.188,A -85,B 0,C 180,E1 18850.201,E2 18850.201} C_VEL
LIN {X 0,Y 508.565,Z 217.173,A -85,B 0,C 180,E1 18849.836,E2 18849.836} C_VEL
LIN {X 0,Y 508.916,Z 223.657,A -85,B 0,C 180,E1 18849.681,E2 18849.681} C_VEL
LIN {X 0,Y 507.779,Z 232.528,A -85,B 0,C 180,E1 18849.637,E2 18849.637} C_VEL
LIN {X 0,Y 504.828,Z 248.226,A -85,B 0,C 180,E1 18849.655,E2 18849.655} C_VEL
LIN {X 0,Y 504.529,Z 252.745,A -85,B 0,C 180,E1 18849.604,E2 18849.604} C_VEL
LIN {X 0,Y 500.335,Z 470.714,A -85,B 0,C 180,E1 18846.062,E2 18846.062} C_VEL
LIN {X 0,Y 499.321,Z 516.581,A -85,B 0,C 180,E1 18845.288,E2 18845.288} C_VEL
LIN {X 0,Y 498.274,Z 537.02,A -85,B 0,C 180,E1 18844.75,E2 18844.75} C_VEL
LIN {X 0,Y 496.904,Z 557.928,A -85,B 0,C 180,E1 18844.002,E2 18844.002} C_VEL
LIN {X 0,Y 495.328,Z 578.017,A -85,B 0,C 180,E1 18843.07,E2 18843.07} C_VEL
LIN {X 0,Y 493.49,Z 597.803,A -85,B 0,C 180,E1 18841.924,E2 18841.924} C_VEL
LIN {X 0,Y 491.516,Z 617.242,A -85,B 0,C 180,E1 18840.567,E2 18840.567} C_VEL
LIN {X 0,Y 489.256,Z 638.981,A -85,B 0,C 180,E1 18838.751,E2 18838.751} C_VEL
LIN {X 0,Y 487.476,Z 656.614,A -85,B 0,C 180,E1 18837.02,E2 18837.02} C_VEL
LIN {X 0,Y 485.786,Z 672.835,A -85,B 0,C 180,E1 18835.151,E2 18835.151} C_VEL
LIN {X 0,Y 484.181,Z 689.073,A -85,B 0,C 180,E1 18832.972,E2 18832.972} C_VEL
LIN {X 0,Y 482.951,Z 702.599,A -85,B 0,C 180,E1 18830.86,E2 18830.86} C_VEL
LIN {X 0,Y 481.885,Z 715.362,A -85,B 0,C 180,E1 18828.509,E2 18828.509} C_VEL
LIN {X 0,Y 481.078,Z 726.642,A -85,B 0,C 180,E1 18826.046,E2 18826.046} C_VEL
LIN {X 0,Y 480.54,Z 736.019,A -85,B 0,C 180,E1 18823.598,E2 18823.598} C_VEL
LIN {X 0,Y 480.201,Z 743.604,A -85,B 0,C 180,E1 18821.165,E2 18821.165} C_VEL
LIN {X 0,Y 480.013,Z 749.806,A -85,B 0,C 180,E1 18818.625,E2 18818.625} C_VEL
LIN {X 0,Y 479.945,Z 754.421,A -85,B 0,C 180,E1 18816.099,E2 18816.099} C_VEL
LIN {X 0,Y 479.913,Z 757.358,A -85,B 0,C 180,E1 18813.583,E2 18813.583} C_VEL
LIN {X 0,Y 479.91,Z 758.815,A -85,B 0,C 180,E1 18810.955,E2 18810.955} C_VEL
LIN {X 0,Y 479.905,Z 758.721,A -85,B 0,C 180,E1 18808.448,E2 18808.448} C_VEL
LIN {X 0,Y 479.918,Z 756.99,A -85,B 0,C 180,E1 18805.938,E2 18805.938} C_VEL
LIN {X 0,Y 479.951,Z 753.595,A -85,B 0,C 180,E1 18803.301,E2 18803.301} C_VEL
LIN {X 0,Y 480.046,Z 748.883,A -85,B 0,C 180,E1 18800.847,E2 18800.847} C_VEL
LIN {X 0,Y 480.249,Z 742.452,A -85,B 0,C 180,E1 18798.349,E2 18798.349} C_VEL
LIN {X 0,Y 480.611,Z 734.644,A -85,B 0,C 180,E1 18795.913,E2 18795.913} C_VEL
LIN {X 0,Y 481.185,Z 724.956,A -85,B 0,C 180,E1 18793.461,E2 18793.461} C_VEL
LIN {X 0,Y 482.011,Z 713.652,A -85,B 0,C 180,E1 18791.068,E2 18791.068} C_VEL
LIN {X 0,Y 483.103,Z 700.869,A -85,B 0,C 180,E1 18788.766,E2 18788.766} C_VEL
LIN {X 0,Y 484.385,Z 687.124,A -85,B 0,C 180,E1 18786.652,E2 18786.652} C_VEL
LIN {X 0,Y 485.918,Z 671.529,A -85,B 0,C 180,E1 18784.598,E2 18784.598} C_VEL
LIN {X 0,Y 487.683,Z 654.406,A -85,B 0,C 180,E1 18782.662,E2 18782.662} C_VEL
LIN {X 0,Y 489.516,Z 636.73,A -85,B 0,C 180,E1 18780.952,E2 18780.952} C_VEL
LIN {X 0,Y 491.85,Z 614.233,A -85,B 0,C 180,E1 18779.111,E2 18779.111} C_VEL
LIN {X 0,Y 493.751,Z 595.192,A -85,B 0,C 180,E1 18777.821,E2 18777.821} C_VEL
LIN {X 0,Y 495.618,Z 574.254,A -85,B 0,C 180,E1 18776.652,E2 18776.652} C_VEL
LIN {X 0,Y 497.258,Z 553.501,A -85,B 0,C 180,E1 18775.73,E2 18775.73} C_VEL
LIN {X 0,Y 498.47,Z 533.571,A -85,B 0,C 180,E1 18775.056,E2 18775.056} C_VEL
LIN {X 0,Y 499.484,Z 510.888,A -85,B 0,C 180,E1 18774.512,E2 18774.512} C_VEL
LIN {X 0,Y 502.843,Z 341.432,A -85,B 0,C 180,E1 18771.744,E2 18771.744} C_VEL
LIN {X 0,Y 504.767,Z 231.825,A -85,B 0,C 180,E1 18769.948,E2 18769.948} C_VEL
LIN {X 0,Y 500.497,Z 205.733,A -85,B 0,C 180,E1 18768.984,E2 18768.984} C_VEL
LIN {X 0,Y 501.876,Z 186.312,A -85,B 0,C 180,E1 18767.488,E2 18767.488} C_VEL
LIN {X 0,Y 494.917,Z 170.787,A -85,B 0,C 180,E1 18765.327,E2 18765.327} C_VEL
LIN {X 0,Y 487.327,Z 155.293,A -85,B 0,C 180,E1 18762.935,E2 18762.935} C_VEL
LIN {X 0,Y 484.682,Z 150.347,A -85,B 0,C 180,E1 18762.102,E2 18762.102} C_VEL
LIN {X 0,Y 482.491,Z 146.119,A -85,B 0,C 180,E1 18761.381,E2 18761.381} C_VEL
LIN {X 0,Y 480.929,Z 142.493,A -85,B 0,C 180,E1 18760.754,E2 18760.754} C_VEL
LIN {X 0,Y 480.831,Z 142.121,A -85,B 0,C 180,E1 18760.259,E2 18760.259} C_VEL
LIN {X 0,Y 480.866,Z 142.123,A -85,B 0,C 180,E1 18756.787,E2 18756.787} C_VEL
LIN {X 0,Y 480.831,Z 142.155,A -85,B 0,C 180,E1 18753.289,E2 18753.289} C_VEL
LIN {X 0,Y 480.819,Z 142.131,A -85,B 0,C 180,E1 18749.802,E2 18749.802} C_VEL
LIN {X 0,Y 480.858,Z 142.124,A -85,B 0,C 180,E1 18746.422,E2 18746.422} C_VEL
LIN {X 0,Y 480.877,Z 142.145,A -85,B 0,C 180,E1 18742.881,E2 18742.881} C_VEL
LIN {X 0,Y 480.833,Z 142.114,A -85,B 0,C 180,E1 18739.433,E2 18739.433} C_VEL
LIN {X 0,Y 480.834,Z 142.152,A -85,B 0,C 180,E1 18735.808,E2 18735.808} C_VEL
LIN {X 0,Y 480.868,Z 142.148,A -85,B 0,C 180,E1 18732.367,E2 18732.367} C_VEL
LIN {X 0,Y 480.893,Z 142.145,A -85,B 0,C 180,E1 18728.73,E2 18728.73} C_VEL
LIN {X 0,Y 480.861,Z 142.151,A -85,B 0,C 180,E1 18725.249,E2 18725.249} C_VEL
LIN {X 0,Y 480.847,Z 142.15,A -85,B 0,C 180,E1 18721.668,E2 18721.668} C_VEL
LIN {X 0,Y 480.86,Z 142.147,A -85,B 0,C 180,E1 18718.094,E2 18718.094} C_VEL
LIN {X 0,Y 480.889,Z 142.144,A -85,B 0,C 180,E1 18714.512,E2 18714.512} C_VEL
LIN {X 0,Y 480.892,Z 142.143,A -85,B 0,C 180,E1 18710.908,E2 18710.908} C_VEL
LIN {X 0,Y 480.874,Z 142.144,A -85,B 0,C 180,E1 18707.268,E2 18707.268} C_VEL
LIN {X 0,Y 480.858,Z 142.117,A -85,B 0,C 180,E1 18703.698,E2 18703.698} C_VEL
LIN {X 0,Y 480.878,Z 142.138,A -85,B 0,C 180,E1 18700.189,E2 18700.189} C_VEL
LIN {X 0,Y 480.891,Z 142.133,A -85,B 0,C 180,E1 18696.602,E2 18696.602} C_VEL
LIN {X 0,Y 480.884,Z 142.113,A -85,B 0,C 180,E1 18693.047,E2 18693.047} C_VEL
LIN {X 0,Y 480.876,Z 142.142,A -85,B 0,C 180,E1 18689.514,E2 18689.514} C_VEL
LIN {X 0,Y 480.875,Z 142.143,A -85,B 0,C 180,E1 18685.845,E2 18685.845} C_VEL
LIN {X 0,Y 480.886,Z 142.122,A -85,B 0,C 180,E1 18682.192,E2 18682.192} C_VEL
LIN {X 0,Y 480.922,Z 142.447,A -85,B 0,C 180,E1 18681.565,E2 18681.565} C_VEL
LIN {X 0,Y 482.474,Z 146.018,A -85,B 0,C 180,E1 18680.95,E2 18680.95} C_VEL
LIN {X 0,Y 483.645,Z 147.984,A -85,B 0,C 180,E1 18680.605,E2 18680.605} C_VEL
LIN {X 0,Y 490.523,Z 161.106,A -85,B 0,C 180,E1 18678.512,E2 18678.512} C_VEL
LIN {X 0,Y 493.184,Z 166.211,A -85,B 0,C 180,E1 18677.793,E2 18677.793} C_VEL
LIN {X 0,Y 507.388,Z 187.37,A -85,B 0,C 180,E1 18675.786,E2 18675.786} C_VEL
LIN {X 0,Y 509.675,Z 191.187,A -85,B 0,C 180,E1 18675.473,E2 18675.473} C_VEL
LIN {X 0,Y 505.566,Z 395.863,A -85,B 0,C 180,E1 18672.047,E2 18672.047} C_VEL
LIN {X 0,Y 503.434,Z 512.151,A -85,B 0,C 180,E1 18670.143,E2 18670.143} C_VEL
LIN {X 0,Y 502.407,Z 534.805,A -85,B 0,C 180,E1 18669.586,E2 18669.586} C_VEL
LIN {X 0,Y 501.151,Z 556.617,A -85,B 0,C 180,E1 18668.869,E2 18668.869} C_VEL
LIN {X 0,Y 499.489,Z 578.896,A -85,B 0,C 180,E1 18667.917,E2 18667.917} C_VEL
LIN {X 0,Y 497.711,Z 600.719,A -85,B 0,C 180,E1 18666.772,E2 18666.772} C_VEL
LIN {X 0,Y 495.818,Z 619.138,A -85,B 0,C 180,E1 18665.575,E2 18665.575} C_VEL
LIN {X 0,Y 493.621,Z 639.175,A -85,B 0,C 180,E1 18664.06,E2 18664.06} C_VEL
LIN {X 0,Y 491.39,Z 658.269,A -85,B 0,C 180,E1 18662.352,E2 18662.352} C_VEL
LIN {X 0,Y 489.088,Z 677.79,A -85,B 0,C 180,E1 18660.327,E2 18660.327} C_VEL
LIN {X 0,Y 487.197,Z 694.156,A -85,B 0,C 180,E1 18658.365,E2 18658.365} C_VEL
LIN {X 0,Y 485.371,Z 710.143,A -85,B 0,C 180,E1 18656.157,E2 18656.157} C_VEL
LIN {X 0,Y 483.888,Z 724.51,A -85,B 0,C 180,E1 18653.89,E2 18653.89} C_VEL
LIN {X 0,Y 482.624,Z 737.451,A -85,B 0,C 180,E1 18651.511,E2 18651.511} C_VEL
LIN {X 0,Y 481.599,Z 749.772,A -85,B 0,C 180,E1 18648.897,E2 18648.897} C_VEL
LIN {X 0,Y 480.908,Z 759.608,A -85,B 0,C 180,E1 18646.424,E2 18646.424} C_VEL
LIN {X 0,Y 480.41,Z 768.994,A -85,B 0,C 180,E1 18643.602,E2 18643.602} C_VEL
LIN {X 0,Y 480.144,Z 775.563,A -85,B 0,C 180,E1 18641.166,E2 18641.166} C_VEL
LIN {X 0,Y 479.98,Z 781.542,A -85,B 0,C 180,E1 18638.318,E2 18638.318} C_VEL
LIN {X 0,Y 479.929,Z 785.119,A -85,B 0,C 180,E1 18635.979,E2 18635.979} C_VEL
LIN {X 0,Y 479.91,Z 787.85,A -85,B 0,C 180,E1 18633.225,E2 18633.225} C_VEL
LIN {X 0,Y 479.901,Z 788.872,A -85,B 0,C 180,E1 18630.716,E2 18630.716} C_VEL
LIN {X 0,Y 479.907,Z 788.527,A -85,B 0,C 180,E1 18627.97,E2 18627.97} C_VEL
LIN {X 0,Y 479.903,Z 786.728,A -85,B 0,C 180,E1 18625.459,E2 18625.459} C_VEL
LIN {X 0,Y 479.958,Z 783.494,A -85,B 0,C 180,E1 18622.82,E2 18622.82} C_VEL
LIN {X 0,Y 480.033,Z 778.828,A -85,B 0,C 180,E1 18620.287,E2 18620.287} C_VEL
LIN {X 0,Y 480.246,Z 772.827,A -85,B 0,C 180,E1 18617.74,E2 18617.74} C_VEL
LIN {X 0,Y 480.616,Z 764.747,A -85,B 0,C 180,E1 18615.051,E2 18615.051} C_VEL
LIN {X 0,Y 481.198,Z 755.447,A -85,B 0,C 180,E1 18612.466,E2 18612.466} C_VEL
LIN {X 0,Y 482.051,Z 744.153,A -85,B 0,C 180,E1 18609.861,E2 18609.861} C_VEL
LIN {X 0,Y 483.249,Z 730.855,A -85,B 0,C 180,E1 18607.238,E2 18607.238} C_VEL
LIN {X 0,Y 484.627,Z 717.221,A -85,B 0,C 180,E1 18604.92,E2 18604.92} C_VEL
LIN {X 0,Y 486.307,Z 701.748,A -85,B 0,C 180,E1 18602.648,E2 18602.648} C_VEL
LIN {X 0,Y 488.285,Z 684.932,A -85,B 0,C 180,E1 18600.49,E2 18600.49} C_VEL
LIN {X 0,Y 490.33,Z 667.178,A -85,B 0,C 180,E1 18598.533,E2 18598.533} C_VEL
LIN {X 0,Y 492.683,Z 647.259,A -85,B 0,C 180,E1 18596.636,E2 18596.636} C_VEL
LIN {X 0,Y 494.769,Z 628.71,A -85,B 0,C 180,E1 18595.118,E2 18595.118} C_VEL
LIN {X 0,Y 496.993,Z 607.836,A -85,B 0,C 180,E1 18593.668,E2 18593.668} C_VEL
LIN {X 0,Y 498.484,Z 591.487,A -85,B 0,C 180,E1 18592.718,E2 18592.718} C_VEL
LIN {X 0,Y 500.268,Z 569.221,A -85,B 0,C 180,E1 18591.643,E2 18591.643} C_VEL
LIN {X 0,Y 501.643,Z 548.02,A -85,B 0,C 180,E1 18590.827,E2 18590.827} C_VEL
LIN {X 0,Y 502.937,Z 523.508,A -85,B 0,C 180,E1 18590.112,E2 18590.112} C_VEL
LIN {X 0,Y 503.753,Z 501.051,A -85,B 0,C 180,E1 18589.656,E2 18589.656} C_VEL
LIN {X 0,Y 507.447,Z 295.86,A -85,B 0,C 180,E1 18586.299,E2 18586.299} C_VEL
LIN {X 0,Y 509.563,Z 190.682,A -85,B 0,C 180,E1 18584.51,E2 18584.51} C_VEL
LIN {X 0,Y 494.415,Z 168.009,A -85,B 0,C 180,E1 18582.391,E2 18582.391} C_VEL
LIN {X 0,Y 492.295,Z 164.487,A -85,B 0,C 180,E1 18582.006,E2 18582.006} C_VEL
LIN {X 0,Y 485.133,Z 150.828,A -85,B 0,C 180,E1 18579.864,E2 18579.864} C_VEL
LIN {X 0,Y 482.901,Z 146.533,A -85,B 0,C 180,E1 18579.161,E2 18579.161} C_VEL
LIN {X 0,Y 481.061,Z 143.094,A -85,B 0,C 180,E1 18578.574,E2 18578.574} C_VEL
LIN {X 0,Y 480.88,Z 142.167,A -85,B 0,C 180,E1 18578.287,E2 18578.287} C_VEL
LIN {X 0,Y 480.887,Z 142.149,A -85,B 0,C 180,E1 18574.729,E2 18574.729} C_VEL
LIN {X 0,Y 480.89,Z 142.129,A -85,B 0,C 180,E1 18571.04,E2 18571.04} C_VEL
LIN {X 0,Y 480.886,Z 142.112,A -85,B 0,C 180,E1 18567.403,E2 18567.403} C_VEL
LIN {X 0,Y 480.884,Z 142.145,A -85,B 0,C 180,E1 18563.789,E2 18563.789} C_VEL
LIN {X 0,Y 480.864,Z 142.128,A -85,B 0,C 180,E1 18560.192,E2 18560.192} C_VEL
LIN {X 0,Y 480.868,Z 142.121,A -85,B 0,C 180,E1 18556.55,E2 18556.55} C_VEL
LIN {X 0,Y 480.888,Z 142.137,A -85,B 0,C 180,E1 18552.976,E2 18552.976} C_VEL
LIN {X 0,Y 480.892,Z 142.139,A -85,B 0,C 180,E1 18549.333,E2 18549.333} C_VEL
LIN {X 0,Y 480.869,Z 142.144,A -85,B 0,C 180,E1 18545.848,E2 18545.848} C_VEL
LIN {X 0,Y 480.853,Z 142.149,A -85,B 0,C 180,E1 18542.264,E2 18542.264} C_VEL
LIN {X 0,Y 480.864,Z 142.148,A -85,B 0,C 180,E1 18538.689,E2 18538.689} C_VEL
LIN {X 0,Y 480.888,Z 142.142,A -85,B 0,C 180,E1 18535.11,E2 18535.11} C_VEL
LIN {X 0,Y 480.871,Z 142.143,A -85,B 0,C 180,E1 18531.631,E2 18531.631} C_VEL
LIN {X 0,Y 480.843,Z 142.148,A -85,B 0,C 180,E1 18528.12,E2 18528.12} C_VEL
LIN {X 0,Y 480.842,Z 142.152,A -85,B 0,C 180,E1 18524.44,E2 18524.44} C_VEL
LIN {X 0,Y 480.866,Z 142.11,A -85,B 0,C 180,E1 18520.946,E2 18520.946} C_VEL
LIN {X 0,Y 480.889,Z 142.149,A -85,B 0,C 180,E1 18517.378,E2 18517.378} C_VEL
LIN {X 0,Y 480.84,Z 142.12,A -85,B 0,C 180,E1 18513.843,E2 18513.843} C_VEL
LIN {X 0,Y 480.825,Z 142.135,A -85,B 0,C 180,E1 18510.336,E2 18510.336} C_VEL
LIN {X 0,Y 480.849,Z 142.152,A -85,B 0,C 180,E1 18506.847,E2 18506.847} C_VEL
LIN {X 0,Y 480.87,Z 142.119,A -85,B 0,C 180,E1 18503.362,E2 18503.362} C_VEL
LIN {X 0,Y 480.819,Z 142.123,A -85,B 0,C 180,E1 18500.017,E2 18500.017} C_VEL
LIN {X 0,Y 480.915,Z 142.404,A -85,B 0,C 180,E1 18499.18,E2 18499.18} C_VEL
LIN {X 0,Y 482.238,Z 145.781,A -85,B 0,C 180,E1 18498.593,E2 18498.593} C_VEL
LIN {X 0,Y 483.392,Z 147.729,A -85,B 0,C 180,E1 18498.238,E2 18498.238} C_VEL
LIN {X 0,Y 490.203,Z 161.065,A -85,B 0,C 180,E1 18496.053,E2 18496.053} C_VEL
LIN {X 0,Y 498.574,Z 178.7,A -85,B 0,C 180,E1 18493.45,E2 18493.45} C_VEL
LIN {X 0,Y 501.956,Z 186.52,A -85,B 0,C 180,E1 18492.395,E2 18492.395} C_VEL
LIN {X 0,Y 500.562,Z 206.662,A -85,B 0,C 180,E1 18490.88,E2 18490.88} C_VEL
LIN {X 0,Y 504.911,Z 233.557,A -85,B 0,C 180,E1 18489.915,E2 18489.915} C_VEL
LIN {X 0,Y 504.529,Z 252.745,A -85,B 0,C 180,E1 18489.604,E2 18489.604} C_VEL
LIN {X 0,Y 503.677,Z 260.446,A -85,B 0,C 180,E1 18489.551,E2 18489.551} C_VEL
LIN {X 0,Y 498.622,Z 281.051,A -85,B 0,C 180,E1 18489.701,E2 18489.701} C_VEL
LIN {X 0,Y 497.928,Z 287.664,A -85,B 0,C 180,E1 18489.653,E2 18489.653} C_VEL
LIN {X 0,Y 493.752,Z 497.127,A -85,B 0,C 180,E1 18486.237,E2 18486.237} C_VEL
LIN {X 0,Y 492.904,Z 522.171,A -85,B 0,C 180,E1 18485.755,E2 18485.755} C_VEL
LIN {X 0,Y 491.751,Z 542.784,A -85,B 0,C 180,E1 18485.171,E2 18485.171} C_VEL
LIN {X 0,Y 490.207,Z 563.383,A -85,B 0,C 180,E1 18484.361,E2 18484.361} C_VEL
LIN {X 0,Y 488.39,Z 583.583,A -85,B 0,C 180,E1 18483.355,E2 18483.355} C_VEL
LIN {X 0,Y 486.42,Z 603.029,A -85,B 0,C 180,E1 18482.166,E2 18482.166} C_VEL
LIN {X 0,Y 484.333,Z 621.497,A -85,B 0,C 180,E1 18480.794,E2 18480.794} C_VEL
LIN {X 0,Y 482.042,Z 640.728,A -85,B 0,C 180,E1 18479.104,E2 18479.104} C_VEL
LIN {X 0,Y 479.899,Z 658.93,A -85,B 0,C 180,E1 18477.214,E2 18477.214} C_VEL
LIN {X 0,Y 478.072,Z 675.373,A -85,B 0,C 180,E1 18475.255,E2 18475.255} C_VEL
LIN {X 0,Y 476.483,Z 690.117,A -85,B 0,C 180,E1 18473.204,E2 18473.204} C_VEL
LIN {X 0,Y 475.107,Z 704.013,A -85,B 0,C 180,E1 18470.962,E2 18470.962} C_VEL
LIN {X 0,Y 473.989,Z 716.635,A -85,B 0,C 180,E1 18468.573,E2 18468.573} C_VEL
LIN {X 0,Y 473.166,Z 727.159,A -85,B 0,C 180,E1 18466.196,E2 18466.196} C_VEL
LIN {X 0,Y 472.559,Z 736.832,A -85,B 0,C 180,E1 18463.583,E2 18463.583} C_VEL
LIN {X 0,Y 472.209,Z 744.312,A -85,B 0,C 180,E1 18461.109,E2 18461.109} C_VEL
LIN {X 0,Y 472.02,Z 750.062,A -85,B 0,C 180,E1 18458.65,E2 18458.65} C_VEL
LIN {X 0,Y 471.945,Z 754.582,A -85,B 0,C 180,E1 18456.081,E2 18456.081} C_VEL
LIN {X 0,Y 471.914,Z 757.358,A -85,B 0,C 180,E1 18453.644,E2 18453.644} C_VEL
LIN {X 0,Y 471.91,Z 758.815,A -85,B 0,C 180,E1 18450.971,E2 18450.971} C_VEL
LIN {X 0,Y 471.904,Z 758.72,A -85,B 0,C 180,E1 18448.422,E2 18448.422} C_VEL
LIN {X 0,Y 471.918,Z 756.989,A -85,B 0,C 180,E1 18445.869,E2 18445.869} C_VEL
LIN {X 0,Y 471.957,Z 753.594,A -85,B 0,C 180,E1 18443.187,E2 18443.187} C_VEL
LIN {X 0,Y 472.059,Z 748.976,A -85,B 0,C 180,E1 18440.737,E2 18440.737} C_VEL
LIN {X 0,Y 472.285,Z 742.45,A -85,B 0,C 180,E1 18438.15,E2 18438.15} C_VEL
LIN {X 0,Y 472.691,Z 734.549,A -85,B 0,C 180,E1 18435.647,E2 18435.647} C_VEL
LIN {X 0,Y 473.317,Z 724.952,A -85,B 0,C 180,E1 18433.178,E2 18433.178} C_VEL
LIN {X 0,Y 474.201,Z 713.908,A -85,B 0,C 180,E1 18430.797,E2 18430.797} C_VEL
LIN {X 0,Y 475.349,Z 701.634,A -85,B 0,C 180,E1 18428.532,E2 18428.532} C_VEL
LIN {X 0,Y 476.816,Z 687.117,A -85,B 0,C 180,E1 18426.259,E2 18426.259} C_VEL
LIN {X 0,Y 478.424,Z 672.009,A -85,B 0,C 180,E1 18424.235,E2 18424.235} C_VEL
LIN {X 0,Y 480.324,Z 655.053,A -85,B 0,C 180,E1 18422.275,E2 18422.275} C_VEL
LIN {X 0,Y 482.453,Z 637.643,A -85,B 0,C 180,E1 18420.509,E2 18420.509} C_VEL
LIN {X 0,Y 484.568,Z 619.387,A -85,B 0,C 180,E1 18418.947,E2 18418.947} C_VEL
LIN {X 0,Y 486.78,Z 599.429,A -85,B 0,C 180,E1 18417.513,E2 18417.513} C_VEL
LIN {X 0,Y 488.806,Z 579.669,A -85,B 0,C 180,E1 18416.336,E2 18416.336} C_VEL
LIN {X 0,Y 490.516,Z 559.435,A -85,B 0,C 180,E1 18415.377,E2 18415.377} C_VEL
LIN {X 0,Y 492.063,Z 537.681,A -85,B 0,C 180,E1 18414.581,E2 18414.581} C_VEL
LIN {X 0,Y 493.146,Z 517.617,A -85,B 0,C 180,E1 18414.046,E2 18414.046} C_VEL
LIN {X 0,Y 494.189,Z 476.117,A -85,B 0,C 180,E1 18413.327,E2 18413.327} C_VEL
LIN {X 0,Y 498.484,Z 259.904,A -85,B 0,C 180,E1 18409.801,E2 18409.801} C_VEL
LIN {X 0,Y 498.879,Z 233.442,A -85,B 0,C 180,E1 18409.349,E2 18409.349} C_VEL
LIN {X 0,Y 494.313,Z 205.093,A -85,B 0,C 180,E1 18408.278,E2 18408.278} C_VEL
LIN {X 0,Y 495.442,Z 190.073,A -85,B 0,C 180,E1 18407.103,E2 18407.103} C_VEL
LIN {X 0,Y 487.385,Z 172.373,A -85,B 0,C 180,E1 18404.556,E2 18404.556} C_VEL
LIN {X 0,Y 481.002,Z 159.496,A -85,B 0,C 180,E1 18402.499,E2 18402.499} C_VEL
LIN {X 0,Y 476.996,Z 151.678,A -85,B 0,C 180,E1 18401.162,E2 18401.162} C_VEL
LIN {X 0,Y 474.896,Z 147.468,A -85,B 0,C 180,E1 18400.427,E2 18400.427} C_VEL
LIN {X 0,Y 473.097,Z 144.241,A -85,B 0,C 180,E1 18399.82,E2 18399.82} C_VEL
LIN {X 0,Y 472.88,Z 143.158,A -85,B 0,C 180,E1 18399.527,E2 18399.527} C_VEL
LIN {X 0,Y 472.873,Z 143.108,A -85,B 0,C 180,E1 18395.852,E2 18395.852} C_VEL
LIN {X 0,Y 472.906,Z 143.124,A -85,B 0,C 180,E1 18392.338,E2 18392.338} C_VEL
LIN {X 0,Y 472.937,Z 143.131,A -85,B 0,C 180,E1 18388.818,E2 18388.818} C_VEL
LIN {X 0,Y 472.896,Z 143.102,A -85,B 0,C 180,E1 18385.284,E2 18385.284} C_VEL
LIN {X 0,Y 472.889,Z 143.141,A -85,B 0,C 180,E1 18381.717,E2 18381.717} C_VEL
LIN {X 0,Y 472.902,Z 143.11,A -85,B 0,C 180,E1 18378.108,E2 18378.108} C_VEL
LIN {X 0,Y 472.948,Z 143.126,A -85,B 0,C 180,E1 18374.571,E2 18374.571} C_VEL
LIN {X 0,Y 472.936,Z 143.128,A -85,B 0,C 180,E1 18370.969,E2 18370.969} C_VEL
LIN {X 0,Y 472.91,Z 143.131,A -85,B 0,C 180,E1 18367.41,E2 18367.41} C_VEL
LIN {X 0,Y 472.906,Z 143.128,A -85,B 0,C 180,E1 18363.758,E2 18363.758} C_VEL
LIN {X 0,Y 472.922,Z 143.127,A -85,B 0,C 180,E1 18360.182,E2 18360.182} C_VEL
LIN {X 0,Y 472.951,Z 143.125,A -85,B 0,C 180,E1 18356.607,E2 18356.607} C_VEL
LIN {X 0,Y 472.953,Z 143.125,A -85,B 0,C 180,E1 18352.957,E2 18352.957} C_VEL
LIN {X 0,Y 472.925,Z 143.127,A -85,B 0,C 180,E1 18349.401,E2 18349.401} C_VEL
LIN {X 0,Y 472.919,Z 143.107,A -85,B 0,C 180,E1 18345.804,E2 18345.804} C_VEL
LIN {X 0,Y 472.937,Z 143.134,A -85,B 0,C 180,E1 18342.149,E2 18342.149} C_VEL
LIN {X 0,Y 472.95,Z 143.094,A -85,B 0,C 180,E1 18338.547,E2 18338.547} C_VEL
LIN {X 0,Y 472.952,Z 143.13,A -85,B 0,C 180,E1 18334.854,E2 18334.854} C_VEL
LIN {X 0,Y 472.949,Z 143.119,A -85,B 0,C 180,E1 18331.183,E2 18331.183} C_VEL
LIN {X 0,Y 472.931,Z 143.102,A -85,B 0,C 180,E1 18327.664,E2 18327.664} C_VEL
LIN {X 0,Y 472.939,Z 143.109,A -85,B 0,C 180,E1 18324.004,E2 18324.004} C_VEL
LIN {X 0,Y 472.986,Z 143.399,A -85,B 0,C 180,E1 18322.649,E2 18322.649} C_VEL
LIN {X 0,Y 474.527,Z 146.991,A -85,B 0,C 180,E1 18322.001,E2 18322.001} C_VEL
LIN {X 0,Y 475.633,Z 148.685,A -85,B 0,C 180,E1 18321.674,E2 18321.674} C_VEL
LIN {X 0,Y 482.728,Z 162.107,A -85,B 0,C 180,E1 18319.43,E2 18319.43} C_VEL
LIN {X 0,Y 485.253,Z 166.877,A -85,B 0,C 180,E1 18318.73,E2 18318.73} C_VEL
LIN {X 0,Y 499.126,Z 187.362,A -85,B 0,C 180,E1 18316.678,E2 18316.678} C_VEL
LIN {X 0,Y 503.709,Z 194.729,A -85,B 0,C 180,E1 18316.03,E2 18316.03} C_VEL
LIN {X 0,Y 499.197,Z 401.266,A -85,B 0,C 180,E1 18312.53,E2 18312.53} C_VEL
LIN {X 0,Y 496.933,Z 512.428,A -85,B 0,C 180,E1 18310.678,E2 18310.678} C_VEL
LIN {X 0,Y 495.839,Z 534.878,A -85,B 0,C 180,E1 18310.117,E2 18310.117} C_VEL
LIN {X 0,Y 494.474,Z 557.129,A -85,B 0,C 180,E1 18309.376,E2 18309.376} C_VEL
LIN {X 0,Y 492.763,Z 578.637,A -85,B 0,C 180,E1 18308.443,E2 18308.443} C_VEL
LIN {X 0,Y 490.873,Z 600.317,A -85,B 0,C 180,E1 18307.298,E2 18307.298} C_VEL
LIN {X 0,Y 488.869,Z 620.365,A -85,B 0,C 180,E1 18306.015,E2 18306.015} C_VEL
LIN {X 0,Y 486.917,Z 638.436,A -85,B 0,C 180,E1 18304.666,E2 18304.666} C_VEL
LIN {X 0,Y 484.478,Z 657.599,A -85,B 0,C 180,E1 18302.942,E2 18302.942} C_VEL
LIN {X 0,Y 482.083,Z 676.679,A -85,B 0,C 180,E1 18300.954,E2 18300.954} C_VEL
LIN {X 0,Y 479.99,Z 693.133,A -85,B 0,C 180,E1 18298.968,E2 18298.968} C_VEL
LIN {X 0,Y 478.009,Z 709.296,A -85,B 0,C 180,E1 18296.725,E2 18296.725} C_VEL
LIN {X 0,Y 476.315,Z 724.172,A -85,B 0,C 180,E1 18294.352,E2 18294.352} C_VEL
LIN {X 0,Y 474.9,Z 737.449,A -85,B 0,C 180,E1 18291.879,E2 18291.879} C_VEL
LIN {X 0,Y 473.831,Z 749.252,A -85,B 0,C 180,E1 18289.347,E2 18289.347} C_VEL
LIN {X 0,Y 473.036,Z 759.399,A -85,B 0,C 180,E1 18286.763,E2 18286.763} C_VEL
LIN {X 0,Y 472.479,Z 768.639,A -85,B 0,C 180,E1 18283.96,E2 18283.96} C_VEL
LIN {X 0,Y 472.182,Z 775.26,A -85,B 0,C 180,E1 18281.481,E2 18281.481} C_VEL
LIN {X 0,Y 471.989,Z 781.222,A -85,B 0,C 180,E1 18278.65,E2 18278.65} C_VEL
LIN {X 0,Y 471.933,Z 784.96,A -85,B 0,C 180,E1 18276.203,E2 18276.203} C_VEL
LIN {X 0,Y 471.91,Z 787.714,A -85,B 0,C 180,E1 18273.523,E2 18273.523} C_VEL
LIN {X 0,Y 471.907,Z 788.849,A -85,B 0,C 180,E1 18270.85,E2 18270.85} C_VEL
LIN {X 0,Y 471.903,Z 788.658,A -85,B 0,C 180,E1 18268.179,E2 18268.179} C_VEL
LIN {X 0,Y 471.903,Z 786.842,A -85,B 0,C 180,E1 18265.504,E2 18265.504} C_VEL
LIN {X 0,Y 471.96,Z 783.681,A -85,B 0,C 180,E1 18262.82,E2 18262.82} C_VEL
LIN {X 0,Y 472.048,Z 778.828,A -85,B 0,C 180,E1 18260.121,E2 18260.121} C_VEL
LIN {X 0,Y 472.283,Z 772.828,A -85,B 0,C 180,E1 18257.53,E2 18257.53} C_VEL
LIN {X 0,Y 472.69,Z 764.746,A -85,B 0,C 180,E1 18254.794,E2 18254.794} C_VEL
LIN {X 0,Y 473.336,Z 755.447,A -85,B 0,C 180,E1 18252.165,E2 18252.165} C_VEL
LIN {X 0,Y 474.218,Z 744.724,A -85,B 0,C 180,E1 18249.642,E2 18249.642} C_VEL
LIN {X 0,Y 475.459,Z 732.14,A -85,B 0,C 180,E1 18247.084,E2 18247.084} C_VEL
LIN {X 0,Y 476.952,Z 718.346,A -85,B 0,C 180,E1 18244.682,E2 18244.682} C_VEL
LIN {X 0,Y 478.858,Z 702.188,A -85,B 0,C 180,E1 18242.25,E2 18242.25} C_VEL
LIN {X 0,Y 480.979,Z 685.537,A -85,B 0,C 180,E1 18240.073,E2 18240.073} C_VEL
LIN {X 0,Y 483.198,Z 667.723,A -85,B 0,C 180,E1 18238.077,E2 18238.077} C_VEL
LIN {X 0,Y 485.626,Z 648.725,A -85,B 0,C 180,E1 18236.228,E2 18236.228} C_VEL
LIN {X 0,Y 487.635,Z 631.873,A -85,B 0,C 180,E1 18234.82,E2 18234.82} C_VEL
LIN {X 0,Y 489.752,Z 611.85,A -85,B 0,C 180,E1 18233.408,E2 18233.408} C_VEL
LIN {X 0,Y 491.71,Z 591.047,A -85,B 0,C 180,E1 18232.189,E2 18232.189} C_VEL
LIN {X 0,Y 493.591,Z 568.708,A -85,B 0,C 180,E1 18231.101,E2 18231.101} C_VEL
LIN {X 0,Y 495.075,Z 547.262,A -85,B 0,C 180,E1 18230.271,E2 18230.271} C_VEL
LIN {X 0,Y 496.44,Z 523.094,A -85,B 0,C 180,E1 18229.566,E2 18229.566} C_VEL
LIN {X 0,Y 497.301,Z 500.489,A -85,B 0,C 180,E1 18229.103,E2 18229.103} C_VEL
LIN {X 0,Y 501.025,Z 311.064,A -85,B 0,C 180,E1 18225.961,E2 18225.961} C_VEL
LIN {X 0,Y 503.567,Z 194.204,A -85,B 0,C 180,E1 18223.943,E2 18223.943} C_VEL
LIN {X 0,Y 489.685,Z 173.318,A -85,B 0,C 180,E1 18221.947,E2 18221.947} C_VEL
LIN {X 0,Y 484.663,Z 165.797,A -85,B 0,C 180,E1 18221.151,E2 18221.151} C_VEL
LIN {X 0,Y 479.01,Z 155.301,A -85,B 0,C 180,E1 18219.44,E2 18219.44} C_VEL
LIN {X 0,Y 477.443,Z 152.141,A -85,B 0,C 180,E1 18218.921,E2 18218.921} C_VEL
LIN {X 0,Y 474.857,Z 147.399,A -85,B 0,C 180,E1 18218.093,E2 18218.093} C_VEL
LIN {X 0,Y 473.074,Z 143.848,A -85,B 0,C 180,E1 18217.466,E2 18217.466} C_VEL
LIN {X 0,Y 472.947,Z 143.137,A -85,B 0,C 180,E1 18217.156,E2 18217.156} C_VEL
LIN {X 0,Y 472.947,Z 143.111,A -85,B 0,C 180,E1 18213.489,E2 18213.489} C_VEL
LIN {X 0,Y 472.951,Z 143.136,A -85,B 0,C 180,E1 18209.789,E2 18209.789} C_VEL
LIN {X 0,Y 472.929,Z 143.11,A -85,B 0,C 180,E1 18206.223,E2 18206.223} C_VEL
LIN {X 0,Y 472.934,Z 143.105,A -85,B 0,C 180,E1 18202.63,E2 18202.63} C_VEL
LIN {X 0,Y 472.951,Z 143.132,A -85,B 0,C 180,E1 18199,E2 18199} C_VEL
LIN {X 0,Y 472.951,Z 143.091,A -85,B 0,C 180,E1 18195.323,E2 18195.323} C_VEL
LIN {X 0,Y 472.941,Z 143.134,A -85,B 0,C 180,E1 18191.71,E2 18191.71} C_VEL
LIN {X 0,Y 472.92,Z 143.135,A -85,B 0,C 180,E1 18188.143,E2 18188.143} C_VEL
LIN {X 0,Y 472.92,Z 143.134,A -85,B 0,C 180,E1 18184.486,E2 18184.486} C_VEL
LIN {X 0,Y 472.937,Z 143.133,A -85,B 0,C 180,E1 18180.848,E2 18180.848} C_VEL
LIN {X 0,Y 472.954,Z 143.132,A -85,B 0,C 180,E1 18177.213,E2 18177.213} C_VEL
LIN {X 0,Y 472.945,Z 143.133,A -85,B 0,C 180,E1 18173.516,E2 18173.516} C_VEL
LIN {X 0,Y 472.91,Z 143.136,A -85,B 0,C 180,E1 18170.016,E2 18170.016} C_VEL
LIN {X 0,Y 472.904,Z 143.134,A -85,B 0,C 180,E1 18166.427,E2 18166.427} C_VEL
LIN {X 0,Y 472.929,Z 143.127,A -85,B 0,C 180,E1 18162.91,E2 18162.91} C_VEL
LIN {X 0,Y 472.946,Z 143.111,A -85,B 0,C 180,E1 18159.326,E2 18159.326} C_VEL
LIN {X 0,Y 472.9,Z 143.117,A -85,B 0,C 180,E1 18155.917,E2 18155.917} C_VEL
LIN {X 0,Y 472.891,Z 143.142,A -85,B 0,C 180,E1 18152.279,E2 18152.279} C_VEL
LIN {X 0,Y 472.904,Z 143.105,A -85,B 0,C 180,E1 18148.801,E2 18148.801} C_VEL
LIN {X 0,Y 472.934,Z 143.113,A -85,B 0,C 180,E1 18145.324,E2 18145.324} C_VEL
LIN {X 0,Y 472.89,Z 143.146,A -85,B 0,C 180,E1 18141.861,E2 18141.861} C_VEL
LIN {X 0,Y 472.895,Z 143.26,A -85,B 0,C 180,E1 18140.318,E2 18140.318} C_VEL
LIN {X 0,Y 473.197,Z 144.555,A -85,B 0,C 180,E1 18140.033,E2 18140.033} C_VEL
LIN {X 0,Y 475.418,Z 148.34,A -85,B 0,C 180,E1 18139.31,E2 18139.31} C_VEL
LIN {X 0,Y 477.157,Z 151.911,A -85,B 0,C 180,E1 18138.695,E2 18138.695} C_VEL
LIN {X 0,Y 482.644,Z 162.738,A -85,B 0,C 180,E1 18136.871,E2 18136.871} C_VEL
LIN {X 0,Y 490.227,Z 178.399,A -85,B 0,C 180,E1 18134.45,E2 18134.45} C_VEL
LIN {X 0,Y 495.519,Z 190.285,A -85,B 0,C 180,E1 18132.779,E2 18132.779} C_VEL
LIN {X 0,Y 494.371,Z 206.125,A -85,B 0,C 180,E1 18131.577,E2 18131.577} C_VEL
LIN {X 0,Y 499.01,Z 235.091,A -85,B 0,C 180,E1 18130.515,E2 18130.515} C_VEL
LIN {X 0,Y 497.928,Z 287.664,A -85,B 0,C 180,E1 18129.653,E2 18129.653} C_VEL
LIN {X 0,Y 497.049,Z 295.367,A -85,B 0,C 180,E1 18129.604,E2 18129.604} C_VEL
LIN {X 0,Y 492.041,Z 315.974,A -85,B 0,C 180,E1 18129.759,E2 18129.759} C_VEL
LIN {X 0,Y 491.331,Z 322.587,A -85,B 0,C 180,E1 18129.713,E2 18129.713} C_VEL
LIN {X 0,Y 487.305,Z 511.218,A -85,B 0,C 180,E1 18126.607,E2 18126.607} C_VEL
LIN {X 0,Y 486.173,Z 533.886,A -85,B 0,C 180,E1 18126.06,E2 18126.06} C_VEL
LIN {X 0,Y 484.779,Z 554.266,A -85,B 0,C 180,E1 18125.36,E2 18125.36} C_VEL
LIN {X 0,Y 483.02,Z 573.761,A -85,B 0,C 180,E1 18124.481,E2 18124.481} C_VEL
LIN {X 0,Y 480.96,Z 593.876,A -85,B 0,C 180,E1 18123.357,E2 18123.357} C_VEL
LIN {X 0,Y 478.826,Z 612.222,A -85,B 0,C 180,E1 18122.101,E2 18122.101} C_VEL
LIN {X 0,Y 476.383,Z 631.487,A -85,B 0,C 180,E1 18120.525,E2 18120.525} C_VEL
LIN {X 0,Y 474.097,Z 649.271,A -85,B 0,C 180,E1 18118.809,E2 18118.809} C_VEL
LIN {X 0,Y 471.936,Z 665.574,A -85,B 0,C 180,E1 18116.96,E2 18116.96} C_VEL
LIN {X 0,Y 469.842,Z 681.987,A -85,B 0,C 180,E1 18114.785,E2 18114.785} C_VEL
LIN {X 0,Y 468.126,Z 697.249,A -85,B 0,C 180,E1 18112.477,E2 18112.477} C_VEL
LIN {X 0,Y 466.8,Z 710.28,A -85,B 0,C 180,E1 18110.172,E2 18110.172} C_VEL
LIN {X 0,Y 465.728,Z 721.836,A -85,B 0,C 180,E1 18107.749,E2 18107.749} C_VEL
LIN {X 0,Y 464.937,Z 732.016,A -85,B 0,C 180,E1 18105.21,E2 18105.21} C_VEL
LIN {X 0,Y 464.435,Z 740.426,A -85,B 0,C 180,E1 18102.685,E2 18102.685} C_VEL
LIN {X 0,Y 464.123,Z 747.257,A -85,B 0,C 180,E1 18100.096,E2 18100.096} C_VEL
LIN {X 0,Y 463.971,Z 752.618,A -85,B 0,C 180,E1 18097.429,E2 18097.429} C_VEL
LIN {X 0,Y 463.921,Z 756.331,A -85,B 0,C 180,E1 18094.821,E2 18094.821} C_VEL
LIN {X 0,Y 463.909,Z 758.355,A -85,B 0,C 180,E1 18092.223,E2 18092.223} C_VEL
LIN {X 0,Y 463.9,Z 758.922,A -85,B 0,C 180,E1 18089.506,E2 18089.506} C_VEL
LIN {X 0,Y 463.91,Z 757.999,A -85,B 0,C 180,E1 18087.035,E2 18087.035} C_VEL
LIN {X 0,Y 463.93,Z 755.498,A -85,B 0,C 180,E1 18084.435,E2 18084.435} C_VEL
LIN {X 0,Y 464.013,Z 751.515,A -85,B 0,C 180,E1 18081.824,E2 18081.824} C_VEL
LIN {X 0,Y 464.18,Z 745.734,A -85,B 0,C 180,E1 18079.186,E2 18079.186} C_VEL
LIN {X 0,Y 464.541,Z 738.339,A -85,B 0,C 180,E1 18076.559,E2 18076.559} C_VEL
LIN {X 0,Y 465.122,Z 729.575,A -85,B 0,C 180,E1 18074.029,E2 18074.029} C_VEL
LIN {X 0,Y 465.987,Z 718.794,A -85,B 0,C 180,E1 18071.485,E2 18071.485} C_VEL
LIN {X 0,Y 467.142,Z 706.599,A -85,B 0,C 180,E1 18069.057,E2 18069.057} C_VEL
LIN {X 0,Y 468.594,Z 693.036,A -85,B 0,C 180,E1 18066.751,E2 18066.751} C_VEL
LIN {X 0,Y 470.575,Z 676.207,A -85,B 0,C 180,E1 18064.314,E2 18064.314} C_VEL
LIN {X 0,Y 472.602,Z 660.562,A -85,B 0,C 180,E1 18062.355,E2 18062.355} C_VEL
LIN {X 0,Y 474.864,Z 643.169,A -85,B 0,C 180,E1 18060.483,E2 18060.483} C_VEL
LIN {X 0,Y 477.229,Z 625.221,A -85,B 0,C 180,E1 18058.836,E2 18058.836} C_VEL
LIN {X 0,Y 479.486,Z 606.613,A -85,B 0,C 180,E1 18057.4,E2 18057.4} C_VEL
LIN {X 0,Y 481.736,Z 586.589,A -85,B 0,C 180,E1 18056.121,E2 18056.121} C_VEL
LIN {X 0,Y 483.741,Z 566.474,A -85,B 0,C 180,E1 18055.074,E2 18055.074} C_VEL
LIN {X 0,Y 485.368,Z 545.734,A -85,B 0,C 180,E1 18054.231,E2 18054.231} C_VEL
LIN {X 0,Y 486.733,Z 524.135,A -85,B 0,C 180,E1 18053.586,E2 18053.586} C_VEL
LIN {X 0,Y 487.621,Z 501.861,A -85,B 0,C 180,E1 18053.133,E2 18053.133} C_VEL
LIN {X 0,Y 491.853,Z 297.794,A -85,B 0,C 180,E1 18049.789,E2 18049.789} C_VEL
LIN {X 0,Y 493.025,Z 234.919,A -85,B 0,C 180,E1 18048.732,E2 18048.732} C_VEL
LIN {X 0,Y 488.193,Z 204.552,A -85,B 0,C 180,E1 18047.559,E2 18047.559} C_VEL
LIN {X 0,Y 489.012,Z 193.889,A -85,B 0,C 180,E1 18046.71,E2 18046.71} C_VEL
LIN {X 0,Y 481.316,Z 176.929,A -85,B 0,C 180,E1 18044.22,E2 18044.22} C_VEL
LIN {X 0,Y 474.073,Z 162.036,A -85,B 0,C 180,E1 18041.795,E2 18041.795} C_VEL
LIN {X 0,Y 469.408,Z 153.087,A -85,B 0,C 180,E1 18040.196,E2 18040.196} C_VEL
LIN {X 0,Y 467.646,Z 149.802,A -85,B 0,C 180,E1 18039.579,E2 18039.579} C_VEL
LIN {X 0,Y 465.18,Z 145.091,A -85,B 0,C 180,E1 18038.678,E2 18038.678} C_VEL
LIN {X 0,Y 464.968,Z 144.15,A -85,B 0,C 180,E1 18038.344,E2 18038.344} C_VEL
LIN {X 0,Y 464.989,Z 144.098,A -85,B 0,C 180,E1 18034.738,E2 18034.738} C_VEL
LIN {X 0,Y 464.96,Z 144.092,A -85,B 0,C 180,E1 18031.147,E2 18031.147} C_VEL
LIN {X 0,Y 464.948,Z 144.131,A -85,B 0,C 180,E1 18027.629,E2 18027.629} C_VEL
LIN {X 0,Y 464.951,Z 144.106,A -85,B 0,C 180,E1 18023.947,E2 18023.947} C_VEL
LIN {X 0,Y 464.993,Z 144.097,A -85,B 0,C 180,E1 18020.518,E2 18020.518} C_VEL
LIN {X 0,Y 465.001,Z 144.116,A -85,B 0,C 180,E1 18016.875,E2 18016.875} C_VEL
LIN {X 0,Y 464.966,Z 144.123,A -85,B 0,C 180,E1 18013.429,E2 18013.429} C_VEL
LIN {X 0,Y 464.964,Z 144.126,A -85,B 0,C 180,E1 18009.781,E2 18009.781} C_VEL
LIN {X 0,Y 464.982,Z 144.127,A -85,B 0,C 180,E1 18006.172,E2 18006.172} C_VEL
LIN {X 0,Y 465.01,Z 144.124,A -85,B 0,C 180,E1 18002.588,E2 18002.588} C_VEL
LIN {X 0,Y 465.014,Z 144.123,A -85,B 0,C 180,E1 17998.891,E2 17998.891} C_VEL
LIN {X 0,Y 464.995,Z 144.125,A -85,B 0,C 180,E1 17995.19,E2 17995.19} C_VEL
LIN {X 0,Y 464.98,Z 144.125,A -85,B 0,C 180,E1 17991.592,E2 17991.592} C_VEL
LIN {X 0,Y 464.982,Z 144.125,A -85,B 0,C 180,E1 17987.835,E2 17987.835} C_VEL
LIN {X 0,Y 464.999,Z 144.08,A -85,B 0,C 180,E1 17984.281,E2 17984.281} C_VEL
LIN {X 0,Y 465.015,Z 144.117,A -85,B 0,C 180,E1 17980.663,E2 17980.663} C_VEL
LIN {X 0,Y 465.015,Z 144.098,A -85,B 0,C 180,E1 17976.962,E2 17976.962} C_VEL
LIN {X 0,Y 464.998,Z 144.089,A -85,B 0,C 180,E1 17973.295,E2 17973.295} C_VEL
LIN {X 0,Y 464.996,Z 144.122,A -85,B 0,C 180,E1 17969.648,E2 17969.648} C_VEL
LIN {X 0,Y 464.999,Z 144.115,A -85,B 0,C 180,E1 17965.875,E2 17965.875} C_VEL
LIN {X 0,Y 465.037,Z 144.38,A -85,B 0,C 180,E1 17963.788,E2 17963.788} C_VEL
LIN {X 0,Y 466.545,Z 147.9,A -85,B 0,C 180,E1 17963.125,E2 17963.125} C_VEL
LIN {X 0,Y 467.724,Z 149.566,A -85,B 0,C 180,E1 17962.773,E2 17962.773} C_VEL
LIN {X 0,Y 469.873,Z 153.551,A -85,B 0,C 180,E1 17962.05,E2 17962.05} C_VEL
LIN {X 0,Y 477.23,Z 167.333,A -85,B 0,C 180,E1 17959.734,E2 17959.734} C_VEL
LIN {X 0,Y 491.622,Z 188.389,A -85,B 0,C 180,E1 17957.509,E2 17957.509} C_VEL
LIN {X 0,Y 497.813,Z 198.219,A -85,B 0,C 180,E1 17956.604,E2 17956.604} C_VEL
LIN {X 0,Y 492.874,Z 404.29,A -85,B 0,C 180,E1 17953.058,E2 17953.058} C_VEL
LIN {X 0,Y 490.459,Z 512.717,A -85,B 0,C 180,E1 17951.224,E2 17951.224} C_VEL
LIN {X 0,Y 489.289,Z 535.22,A -85,B 0,C 180,E1 17950.653,E2 17950.653} C_VEL
LIN {X 0,Y 487.845,Z 557.426,A -85,B 0,C 180,E1 17949.903,E2 17949.903} C_VEL
LIN {X 0,Y 486.032,Z 578.918,A -85,B 0,C 180,E1 17948.957,E2 17948.957} C_VEL
LIN {X 0,Y 483.966,Z 600.946,A -85,B 0,C 180,E1 17947.774,E2 17947.774} C_VEL
LIN {X 0,Y 481.851,Z 620.907,A -85,B 0,C 180,E1 17946.476,E2 17946.476} C_VEL
LIN {X 0,Y 479.333,Z 642.649,A -85,B 0,C 180,E1 17944.805,E2 17944.805} C_VEL
LIN {X 0,Y 477.119,Z 660.924,A -85,B 0,C 180,E1 17943.157,E2 17943.157} C_VEL
LIN {X 0,Y 474.653,Z 678.898,A -85,B 0,C 180,E1 17941.211,E2 17941.211} C_VEL
LIN {X 0,Y 472.402,Z 695.675,A -85,B 0,C 180,E1 17939.13,E2 17939.13} C_VEL
LIN {X 0,Y 470.351,Z 710.985,A -85,B 0,C 180,E1 17936.922,E2 17936.922} C_VEL
LIN {X 0,Y 468.519,Z 725.944,A -85,B 0,C 180,E1 17934.456,E2 17934.456} C_VEL
LIN {X 0,Y 467.062,Z 738.717,A -85,B 0,C 180,E1 17932.001,E2 17932.001} C_VEL
LIN {X 0,Y 465.821,Z 751.325,A -85,B 0,C 180,E1 17929.171,E2 17929.171} C_VEL
LIN {X 0,Y 465.004,Z 761.524,A -85,B 0,C 180,E1 17926.465,E2 17926.465} C_VEL
LIN {X 0,Y 464.463,Z 770.055,A -85,B 0,C 180,E1 17923.697,E2 17923.697} C_VEL
LIN {X 0,Y 464.147,Z 777.045,A -85,B 0,C 180,E1 17920.927,E2 17920.927} C_VEL
LIN {X 0,Y 463.988,Z 782.049,A -85,B 0,C 180,E1 17918.301,E2 17918.301} C_VEL
LIN {X 0,Y 463.919,Z 785.756,A -85,B 0,C 180,E1 17915.69,E2 17915.69} C_VEL
LIN {X 0,Y 463.914,Z 788.053,A -85,B 0,C 180,E1 17912.965,E2 17912.965} C_VEL
LIN {X 0,Y 463.898,Z 788.917,A -85,B 0,C 180,E1 17910.494,E2 17910.494} C_VEL
LIN {X 0,Y 463.907,Z 788.393,A -85,B 0,C 180,E1 17907.653,E2 17907.653} C_VEL
LIN {X 0,Y 463.91,Z 786.614,A -85,B 0,C 180,E1 17905.178,E2 17905.178} C_VEL
LIN {X 0,Y 463.974,Z 783.081,A -85,B 0,C 180,E1 17902.322,E2 17902.322} C_VEL
LIN {X 0,Y 464.08,Z 778.574,A -85,B 0,C 180,E1 17899.825,E2 17899.825} C_VEL
LIN {X 0,Y 464.349,Z 772.172,A -85,B 0,C 180,E1 17897.06,E2 17897.06} C_VEL
LIN {X 0,Y 464.799,Z 764.341,A -85,B 0,C 180,E1 17894.402,E2 17894.402} C_VEL
LIN {X 0,Y 465.574,Z 754.417,A -85,B 0,C 180,E1 17891.598,E2 17891.598} C_VEL
LIN {X 0,Y 466.572,Z 743.576,A -85,B 0,C 180,E1 17889.031,E2 17889.031} C_VEL
LIN {X 0,Y 468.015,Z 730.151,A -85,B 0,C 180,E1 17886.32,E2 17886.32} C_VEL
LIN {X 0,Y 469.741,Z 716.023,A -85,B 0,C 180,E1 17883.858,E2 17883.858} C_VEL
LIN {X 0,Y 471.751,Z 700.335,A -85,B 0,C 180,E1 17881.519,E2 17881.519} C_VEL
LIN {X 0,Y 474.05,Z 683.337,A -85,B 0,C 180,E1 17879.309,E2 17879.309} C_VEL
LIN {X 0,Y 476.349,Z 666.565,A -85,B 0,C 180,E1 17877.427,E2 17877.427} C_VEL
LIN {X 0,Y 478.52,Z 649.758,A -85,B 0,C 180,E1 17875.802,E2 17875.802} C_VEL
LIN {X 0,Y 480.793,Z 630.144,A -85,B 0,C 180,E1 17874.198,E2 17874.198} C_VEL
LIN {X 0,Y 483.216,Z 608.29,A -85,B 0,C 180,E1 17872.681,E2 17872.681} C_VEL
LIN {X 0,Y 485.154,Z 588.864,A -85,B 0,C 180,E1 17871.549,E2 17871.549} C_VEL
LIN {X 0,Y 487.12,Z 565.882,A -85,B 0,C 180,E1 17870.447,E2 17870.447} C_VEL
LIN {X 0,Y 488.82,Z 543.271,A -85,B 0,C 180,E1 17869.589,E2 17869.589} C_VEL
LIN {X 0,Y 490.054,Z 521.079,A -85,B 0,C 180,E1 17868.97,E2 17868.97} C_VEL
LIN {X 0,Y 490.944,Z 497.004,A -85,B 0,C 180,E1 17868.489,E2 17868.489} C_VEL
LIN {X 0,Y 494.924,Z 313.443,A -85,B 0,C 180,E1 17865.394,E2 17865.394} C_VEL
LIN {X 0,Y 497.719,Z 197.811,A -85,B 0,C 180,E1 17863.376,E2 17863.376} C_VEL
LIN {X 0,Y 483.239,Z 175.991,A -85,B 0,C 180,E1 17861.223,E2 17861.223} C_VEL
LIN {X 0,Y 476.479,Z 166.199,A -85,B 0,C 180,E1 17860.107,E2 17860.107} C_VEL
LIN {X 0,Y 471.602,Z 157.102,A -85,B 0,C 180,E1 17858.559,E2 17858.559} C_VEL
LIN {X 0,Y 469.438,Z 153.004,A -85,B 0,C 180,E1 17857.836,E2 17857.836} C_VEL
LIN {X 0,Y 466.938,Z 148.385,A -85,B 0,C 180,E1 17856.992,E2 17856.992} C_VEL
LIN {X 0,Y 465.149,Z 144.938,A -85,B 0,C 180,E1 17856.351,E2 17856.351} C_VEL
LIN {X 0,Y 465.004,Z 144.141,A -85,B 0,C 180,E1 17856.055,E2 17856.055} C_VEL
LIN {X 0,Y 464.993,Z 144.089,A -85,B 0,C 180,E1 17852.325,E2 17852.325} C_VEL
LIN {X 0,Y 465.005,Z 144.102,A -85,B 0,C 180,E1 17848.652,E2 17848.652} C_VEL
LIN {X 0,Y 465.012,Z 144.122,A -85,B 0,C 180,E1 17844.925,E2 17844.925} C_VEL
LIN {X 0,Y 465.01,Z 144.081,A -85,B 0,C 180,E1 17841.308,E2 17841.308} C_VEL
LIN {X 0,Y 465.008,Z 144.117,A -85,B 0,C 180,E1 17837.648,E2 17837.648} C_VEL
LIN {X 0,Y 464.983,Z 144.095,A -85,B 0,C 180,E1 17834.063,E2 17834.063} C_VEL
LIN {X 0,Y 464.985,Z 144.115,A -85,B 0,C 180,E1 17830.406,E2 17830.406} C_VEL
LIN {X 0,Y 464.999,Z 144.115,A -85,B 0,C 180,E1 17826.792,E2 17826.792} C_VEL
LIN {X 0,Y 465.013,Z 144.114,A -85,B 0,C 180,E1 17823.205,E2 17823.205} C_VEL
LIN {X 0,Y 465.011,Z 144.112,A -85,B 0,C 180,E1 17819.507,E2 17819.507} C_VEL
LIN {X 0,Y 464.977,Z 144.116,A -85,B 0,C 180,E1 17815.931,E2 17815.931} C_VEL
LIN {X 0,Y 464.967,Z 144.12,A -85,B 0,C 180,E1 17812.338,E2 17812.338} C_VEL
LIN {X 0,Y 464.98,Z 144.12,A -85,B 0,C 180,E1 17808.715,E2 17808.715} C_VEL
LIN {X 0,Y 465.016,Z 144.115,A -85,B 0,C 180,E1 17805.175,E2 17805.175} C_VEL
LIN {X 0,Y 464.997,Z 144.086,A -85,B 0,C 180,E1 17801.483,E2 17801.483} C_VEL
LIN {X 0,Y 464.964,Z 144.129,A -85,B 0,C 180,E1 17797.894,E2 17797.894} C_VEL
LIN {X 0,Y 464.948,Z 144.091,A -85,B 0,C 180,E1 17794.253,E2 17794.253} C_VEL
LIN {X 0,Y 464.96,Z 144.114,A -85,B 0,C 180,E1 17790.64,E2 17790.64} C_VEL
LIN {X 0,Y 464.999,Z 144.117,A -85,B 0,C 180,E1 17787.189,E2 17787.189} C_VEL
LIN {X 0,Y 464.976,Z 144.094,A -85,B 0,C 180,E1 17783.534,E2 17783.534} C_VEL
LIN {X 0,Y 465.028,Z 144.38,A -85,B 0,C 180,E1 17781.39,E2 17781.39} C_VEL
LIN {X 0,Y 466.585,Z 148.039,A -85,B 0,C 180,E1 17780.676,E2 17780.676} C_VEL
LIN {X 0,Y 467.758,Z 150.101,A -85,B 0,C 180,E1 17780.273,E2 17780.273} C_VEL
LIN {X 0,Y 470.338,Z 155.002,A -85,B 0,C 180,E1 17779.367,E2 17779.367} C_VEL
LIN {X 0,Y 476.758,Z 167.486,A -85,B 0,C 180,E1 17777.196,E2 17777.196} C_VEL
LIN {X 0,Y 484.999,Z 184.787,A -85,B 0,C 180,E1 17774.496,E2 17774.496} C_VEL
LIN {X 0,Y 489.079,Z 194.074,A -85,B 0,C 180,E1 17773.174,E2 17773.174} C_VEL
LIN {X 0,Y 488.255,Z 205.705,A -85,B 0,C 180,E1 17772.288,E2 17772.288} C_VEL
LIN {X 0,Y 493.161,Z 236.577,A -85,B 0,C 180,E1 17771.129,E2 17771.129} C_VEL
LIN {X 0,Y 491.331,Z 322.587,A -85,B 0,C 180,E1 17769.713,E2 17769.713} C_VEL
LIN {X 0,Y 490.412,Z 330.293,A -85,B 0,C 180,E1 17769.669,E2 17769.669} C_VEL
LIN {X 0,Y 485.379,Z 350.888,A -85,B 0,C 180,E1 17769.834,E2 17769.834} C_VEL
LIN {X 0,Y 484.701,Z 357.497,A -85,B 0,C 180,E1 17769.784,E2 17769.784} C_VEL
LIN {X 0,Y 481.219,Z 514.31,A -85,B 0,C 180,E1 17767.182,E2 17767.182} C_VEL
LIN {X 0,Y 480.042,Z 535.489,A -85,B 0,C 180,E1 17766.645,E2 17766.645} C_VEL
LIN {X 0,Y 478.593,Z 555.431,A -85,B 0,C 180,E1 17765.947,E2 17765.947} C_VEL
LIN {X 0,Y 476.618,Z 575.688,A -85,B 0,C 180,E1 17765.011,E2 17765.011} C_VEL
LIN {X 0,Y 474.302,Z 596.354,A -85,B 0,C 180,E1 17763.815,E2 17763.815} C_VEL
LIN {X 0,Y 471.956,Z 615.325,A -85,B 0,C 180,E1 17762.482,E2 17762.482} C_VEL
LIN {X 0,Y 469.362,Z 634.069,A -85,B 0,C 180,E1 17760.889,E2 17760.889} C_VEL
LIN {X 0,Y 466.741,Z 652.48,A -85,B 0,C 180,E1 17759.032,E2 17759.032} C_VEL
LIN {X 0,Y 464.326,Z 669.458,A -85,B 0,C 180,E1 17757.023,E2 17757.023} C_VEL
LIN {X 0,Y 462.243,Z 684.434,A -85,B 0,C 180,E1 17754.947,E2 17754.947} C_VEL
LIN {X 0,Y 460.434,Z 698.113,A -85,B 0,C 180,E1 17752.739,E2 17752.739} C_VEL
LIN {X 0,Y 458.786,Z 712.828,A -85,B 0,C 180,E1 17750.008,E2 17750.008} C_VEL
LIN {X 0,Y 457.713,Z 724.075,A -85,B 0,C 180,E1 17747.545,E2 17747.545} C_VEL
LIN {X 0,Y 456.912,Z 733.852,A -85,B 0,C 180,E1 17744.964,E2 17744.964} C_VEL
LIN {X 0,Y 456.379,Z 742.196,A -85,B 0,C 180,E1 17742.269,E2 17742.269} C_VEL
LIN {X 0,Y 456.094,Z 748.793,A -85,B 0,C 180,E1 17739.59,E2 17739.59} C_VEL
LIN {X 0,Y 455.97,Z 753.447,A -85,B 0,C 180,E1 17737.053,E2 17737.053} C_VEL
LIN {X 0,Y 455.92,Z 756.904,A -85,B 0,C 180,E1 17734.276,E2 17734.276} C_VEL
LIN {X 0,Y 455.901,Z 758.689,A -85,B 0,C 180,E1 17731.634,E2 17731.634} C_VEL
LIN {X 0,Y 455.912,Z 758.832,A -85,B 0,C 180,E1 17728.995,E2 17728.995} C_VEL
LIN {X 0,Y 455.916,Z 757.441,A -85,B 0,C 180,E1 17726.228,E2 17726.228} C_VEL
LIN {X 0,Y 455.945,Z 754.699,A -85,B 0,C 180,E1 17723.705,E2 17723.705} C_VEL
LIN {X 0,Y 456.041,Z 750.244,A -85,B 0,C 180,E1 17721.045,E2 17721.045} C_VEL
LIN {X 0,Y 456.291,Z 744.212,A -85,B 0,C 180,E1 17718.37,E2 17718.37} C_VEL
LIN {X 0,Y 456.712,Z 736.713,A -85,B 0,C 180,E1 17715.807,E2 17715.807} C_VEL
LIN {X 0,Y 457.436,Z 727.005,A -85,B 0,C 180,E1 17713.1,E2 17713.1} C_VEL
LIN {X 0,Y 458.429,Z 716.44,A -85,B 0,C 180,E1 17710.639,E2 17710.639} C_VEL
LIN {X 0,Y 459.733,Z 704.107,A -85,B 0,C 180,E1 17708.229,E2 17708.229} C_VEL
LIN {X 0,Y 461.508,Z 689.817,A -85,B 0,C 180,E1 17705.797,E2 17705.797} C_VEL
LIN {X 0,Y 463.539,Z 674.987,A -85,B 0,C 180,E1 17703.619,E2 17703.619} C_VEL
LIN {X 0,Y 465.755,Z 659.464,A -85,B 0,C 180,E1 17701.663,E2 17701.663} C_VEL
LIN {X 0,Y 468.18,Z 642.4,A -85,B 0,C 180,E1 17699.822,E2 17699.822} C_VEL
LIN {X 0,Y 470.749,Z 624.135,A -85,B 0,C 180,E1 17698.144,E2 17698.144} C_VEL
LIN {X 0,Y 473.121,Z 606.029,A -85,B 0,C 180,E1 17696.743,E2 17696.743} C_VEL
LIN {X 0,Y 475.468,Z 586.382,A -85,B 0,C 180,E1 17695.486,E2 17695.486} C_VEL
LIN {X 0,Y 477.573,Z 566.503,A -85,B 0,C 180,E1 17694.445,E2 17694.445} C_VEL
LIN {X 0,Y 479.315,Z 545.759,A -85,B 0,C 180,E1 17693.598,E2 17693.598} C_VEL
LIN {X 0,Y 480.732,Z 524.299,A -85,B 0,C 180,E1 17692.956,E2 17692.956} C_VEL
LIN {X 0,Y 481.655,Z 501.68,A -85,B 0,C 180,E1 17692.496,E2 17692.496} C_VEL
LIN {X 0,Y 486.238,Z 286.948,A -85,B 0,C 180,E1 17688.965,E2 17688.965} C_VEL
LIN {X 0,Y 487.246,Z 236.563,A -85,B 0,C 180,E1 17688.107,E2 17688.107} C_VEL
LIN {X 0,Y 482.148,Z 203.962,A -85,B 0,C 180,E1 17686.818,E2 17686.818} C_VEL
LIN {X 0,Y 482.617,Z 197.687,A -85,B 0,C 180,E1 17686.306,E2 17686.306} C_VEL
LIN {X 0,Y 474.401,Z 179.466,A -85,B 0,C 180,E1 17683.566,E2 17683.566} C_VEL
LIN {X 0,Y 466.419,Z 163.355,A -85,B 0,C 180,E1 17680.826,E2 17680.826} C_VEL
LIN {X 0,Y 461.506,Z 154.115,A -85,B 0,C 180,E1 17679.084,E2 17679.084} C_VEL
LIN {X 0,Y 459.143,Z 149.633,A -85,B 0,C 180,E1 17678.204,E2 17678.204} C_VEL
LIN {X 0,Y 457.382,Z 146.757,A -85,B 0,C 180,E1 17677.583,E2 17677.583} C_VEL
LIN {X 0,Y 457.021,Z 145.155,A -85,B 0,C 180,E1 17677.201,E2 17677.201} C_VEL
LIN {X 0,Y 457.002,Z 145.122,A -85,B 0,C 180,E1 17673.61,E2 17673.61} C_VEL
LIN {X 0,Y 457.004,Z 145.088,A -85,B 0,C 180,E1 17669.923,E2 17669.923} C_VEL
LIN {X 0,Y 457.047,Z 145.084,A -85,B 0,C 180,E1 17666.505,E2 17666.505} C_VEL
LIN {X 0,Y 457.069,Z 145.111,A -85,B 0,C 180,E1 17662.78,E2 17662.78} C_VEL
LIN {X 0,Y 457.039,Z 145.07,A -85,B 0,C 180,E1 17659.082,E2 17659.082} C_VEL
LIN {X 0,Y 457.023,Z 145.12,A -85,B 0,C 180,E1 17655.48,E2 17655.48} C_VEL
LIN {X 0,Y 457.023,Z 145.116,A -85,B 0,C 180,E1 17651.74,E2 17651.74} C_VEL
LIN {X 0,Y 457.032,Z 145.111,A -85,B 0,C 180,E1 17648.049,E2 17648.049} C_VEL
LIN {X 0,Y 457.065,Z 145.104,A -85,B 0,C 180,E1 17644.517,E2 17644.517} C_VEL
LIN {X 0,Y 457.08,Z 145.102,A -85,B 0,C 180,E1 17640.752,E2 17640.752} C_VEL
LIN {X 0,Y 457.058,Z 145.106,A -85,B 0,C 180,E1 17637.116,E2 17637.116} C_VEL
LIN {X 0,Y 457.042,Z 145.107,A -85,B 0,C 180,E1 17633.468,E2 17633.468} C_VEL
LIN {X 0,Y 457.04,Z 145.104,A -85,B 0,C 180,E1 17629.793,E2 17629.793} C_VEL
LIN {X 0,Y 457.056,Z 145.086,A -85,B 0,C 180,E1 17626.205,E2 17626.205} C_VEL
LIN {X 0,Y 457.073,Z 145.099,A -85,B 0,C 180,E1 17622.503,E2 17622.503} C_VEL
LIN {X 0,Y 457.071,Z 145.069,A -85,B 0,C 180,E1 17618.842,E2 17618.842} C_VEL
LIN {X 0,Y 457.069,Z 145.113,A -85,B 0,C 180,E1 17615.165,E2 17615.165} C_VEL
LIN {X 0,Y 457.056,Z 145.085,A -85,B 0,C 180,E1 17611.517,E2 17611.517} C_VEL
LIN {X 0,Y 457.054,Z 145.076,A -85,B 0,C 180,E1 17607.842,E2 17607.842} C_VEL
LIN {X 0,Y 457.109,Z 145.37,A -85,B 0,C 180,E1 17604.996,E2 17604.996} C_VEL
LIN {X 0,Y 458.366,Z 148.558,A -85,B 0,C 180,E1 17604.379,E2 17604.379} C_VEL
LIN {X 0,Y 459.88,Z 150.721,A -85,B 0,C 180,E1 17603.9,E2 17603.9} C_VEL
LIN {X 0,Y 461.975,Z 154.538,A -85,B 0,C 180,E1 17603.165,E2 17603.165} C_VEL
LIN {X 0,Y 469.244,Z 168.014,A -85,B 0,C 180,E1 17600.779,E2 17600.779} C_VEL
LIN {X 0,Y 482.461,Z 186.941,A -85,B 0,C 180,E1 17598.636,E2 17598.636} C_VEL
LIN {X 0,Y 491.969,Z 201.893,A -85,B 0,C 180,E1 17597.188,E2 17597.188} C_VEL
LIN {X 0,Y 486.483,Z 411.797,A -85,B 0,C 180,E1 17593.524,E2 17593.524} C_VEL
LIN {X 0,Y 484.026,Z 512.527,A -85,B 0,C 180,E1 17591.79,E2 17591.79} C_VEL
LIN {X 0,Y 482.764,Z 535.329,A -85,B 0,C 180,E1 17591.204,E2 17591.204} C_VEL
LIN {X 0,Y 481.164,Z 558.217,A -85,B 0,C 180,E1 17590.415,E2 17590.415} C_VEL
LIN {X 0,Y 479.251,Z 579.925,A -85,B 0,C 180,E1 17589.447,E2 17589.447} C_VEL
LIN {X 0,Y 476.938,Z 603.013,A -85,B 0,C 180,E1 17588.173,E2 17588.173} C_VEL
LIN {X 0,Y 474.765,Z 622.391,A -85,B 0,C 180,E1 17586.884,E2 17586.884} C_VEL
LIN {X 0,Y 472.225,Z 642.942,A -85,B 0,C 180,E1 17585.269,E2 17585.269} C_VEL
LIN {X 0,Y 469.82,Z 661.755,A -85,B 0,C 180,E1 17583.55,E2 17583.55} C_VEL
LIN {X 0,Y 467.378,Z 679.893,A -85,B 0,C 180,E1 17581.608,E2 17581.608} C_VEL
LIN {X 0,Y 465.409,Z 693.648,A -85,B 0,C 180,E1 17579.894,E2 17579.894} C_VEL
LIN {X 0,Y 463.055,Z 710.138,A -85,B 0,C 180,E1 17577.521,E2 17577.521} C_VEL
LIN {X 0,Y 461.14,Z 724.506,A -85,B 0,C 180,E1 17575.148,E2 17575.148} C_VEL
LIN {X 0,Y 459.517,Z 737.445,A -85,B 0,C 180,E1 17572.651,E2 17572.651} C_VEL
LIN {X 0,Y 458.246,Z 749.255,A -85,B 0,C 180,E1 17570.032,E2 17570.032} C_VEL
LIN {X 0,Y 457.308,Z 759.146,A -85,B 0,C 180,E1 17567.429,E2 17567.429} C_VEL
LIN {X 0,Y 456.629,Z 768.312,A -85,B 0,C 180,E1 17564.574,E2 17564.574} C_VEL
LIN {X 0,Y 456.245,Z 775.259,A -85,B 0,C 180,E1 17561.888,E2 17561.888} C_VEL
LIN {X 0,Y 456.016,Z 781.223,A -85,B 0,C 180,E1 17558.956,E2 17558.956} C_VEL
LIN {X 0,Y 455.941,Z 784.959,A -85,B 0,C 180,E1 17556.421,E2 17556.421} C_VEL
LIN {X 0,Y 455.911,Z 787.713,A -85,B 0,C 180,E1 17553.646,E2 17553.646} C_VEL
LIN {X 0,Y 455.911,Z 788.826,A -85,B 0,C 180,E1 17551.005,E2 17551.005} C_VEL
LIN {X 0,Y 455.901,Z 788.713,A -85,B 0,C 180,E1 17548.366,E2 17548.366} C_VEL
LIN {X 0,Y 455.905,Z 787.069,A -85,B 0,C 180,E1 17545.598,E2 17545.598} C_VEL
LIN {X 0,Y 455.955,Z 784.32,A -85,B 0,C 180,E1 17543.073,E2 17543.073} C_VEL
LIN {X 0,Y 456.061,Z 779.591,A -85,B 0,C 180,E1 17540.154,E2 17540.154} C_VEL
LIN {X 0,Y 456.3,Z 774.046,A -85,B 0,C 180,E1 17537.6,E2 17537.6} C_VEL
LIN {X 0,Y 456.779,Z 765.959,A -85,B 0,C 180,E1 17534.642,E2 17534.642} C_VEL
LIN {X 0,Y 457.465,Z 757.314,A -85,B 0,C 180,E1 17532.051,E2 17532.051} C_VEL
LIN {X 0,Y 458.574,Z 745.868,A -85,B 0,C 180,E1 17529.183,E2 17529.183} C_VEL
LIN {X 0,Y 460.021,Z 733.431,A -85,B 0,C 180,E1 17526.522,E2 17526.522} C_VEL
LIN {X 0,Y 461.796,Z 719.329,A -85,B 0,C 180,E1 17523.966,E2 17523.966} C_VEL
LIN {X 0,Y 464.04,Z 703.11,A -85,B 0,C 180,E1 17521.424,E2 17521.424} C_VEL
LIN {X 0,Y 466.323,Z 687.4,A -85,B 0,C 180,E1 17519.293,E2 17519.293} C_VEL
LIN {X 0,Y 468.657,Z 670.308,A -85,B 0,C 180,E1 17517.333,E2 17517.333} C_VEL
LIN {X 0,Y 471.017,Z 652.612,A -85,B 0,C 180,E1 17515.584,E2 17515.584} C_VEL
LIN {X 0,Y 473.481,Z 632.824,A -85,B 0,C 180,E1 17513.903,E2 17513.903} C_VEL
LIN {X 0,Y 475.857,Z 613.006,A -85,B 0,C 180,E1 17512.459,E2 17512.459} C_VEL
LIN {X 0,Y 478.082,Z 592.172,A -85,B 0,C 180,E1 17511.196,E2 17511.196} C_VEL
LIN {X 0,Y 480.14,Z 570.594,A -85,B 0,C 180,E1 17510.106,E2 17510.106} C_VEL
LIN {X 0,Y 481.87,Z 548.091,A -85,B 0,C 180,E1 17509.21,E2 17509.21} C_VEL
LIN {X 0,Y 483.444,Z 523.75,A -85,B 0,C 180,E1 17508.475,E2 17508.475} C_VEL
LIN {X 0,Y 484.4,Z 501.907,A -85,B 0,C 180,E1 17508.01,E2 17508.01} C_VEL
LIN {X 0,Y 489.282,Z 301.195,A -85,B 0,C 180,E1 17504.556,E2 17504.556} C_VEL
LIN {X 0,Y 491.869,Z 201.471,A -85,B 0,C 180,E1 17502.79,E2 17502.79} C_VEL
LIN {X 0,Y 478.889,Z 181.762,A -85,B 0,C 180,E1 17500.806,E2 17500.806} C_VEL
LIN {X 0,Y 468.805,Z 167.444,A -85,B 0,C 180,E1 17499.146,E2 17499.146} C_VEL
LIN {X 0,Y 463.817,Z 158.227,A -85,B 0,C 180,E1 17497.507,E2 17497.507} C_VEL
LIN {X 0,Y 461.585,Z 154.056,A -85,B 0,C 180,E1 17496.731,E2 17496.731} C_VEL
LIN {X 0,Y 459.129,Z 149.527,A -85,B 0,C 180,E1 17495.86,E2 17495.86} C_VEL
LIN {X 0,Y 457.265,Z 146.126,A -85,B 0,C 180,E1 17495.181,E2 17495.181} C_VEL
LIN {X 0,Y 457.076,Z 145.141,A -85,B 0,C 180,E1 17494.886,E2 17494.886} C_VEL
LIN {X 0,Y 457.073,Z 145.087,A -85,B 0,C 180,E1 17491.081,E2 17491.081} C_VEL
LIN {X 0,Y 457.068,Z 145.072,A -85,B 0,C 180,E1 17487.347,E2 17487.347} C_VEL
LIN {X 0,Y 457.075,Z 145.099,A -85,B 0,C 180,E1 17483.574,E2 17483.574} C_VEL
LIN {X 0,Y 457.062,Z 145.095,A -85,B 0,C 180,E1 17479.82,E2 17479.82} C_VEL
LIN {X 0,Y 457.045,Z 145.073,A -85,B 0,C 180,E1 17476.131,E2 17476.131} C_VEL
LIN {X 0,Y 457.045,Z 145.115,A -85,B 0,C 180,E1 17472.38,E2 17472.38} C_VEL
LIN {X 0,Y 457.056,Z 145.115,A -85,B 0,C 180,E1 17468.681,E2 17468.681} C_VEL
LIN {X 0,Y 457.071,Z 145.116,A -85,B 0,C 180,E1 17465.02,E2 17465.02} C_VEL
LIN {X 0,Y 457.08,Z 145.114,A -85,B 0,C 180,E1 17461.253,E2 17461.253} C_VEL
LIN {X 0,Y 457.061,Z 145.115,A -85,B 0,C 180,E1 17457.618,E2 17457.618} C_VEL
LIN {X 0,Y 457.038,Z 145.116,A -85,B 0,C 180,E1 17453.972,E2 17453.972} C_VEL
LIN {X 0,Y 457.029,Z 145.115,A -85,B 0,C 180,E1 17450.302,E2 17450.302} C_VEL
LIN {X 0,Y 457.033,Z 145.112,A -85,B 0,C 180,E1 17446.591,E2 17446.591} C_VEL
LIN {X 0,Y 457.065,Z 145.105,A -85,B 0,C 180,E1 17443.085,E2 17443.085} C_VEL
LIN {X 0,Y 457.064,Z 145.083,A -85,B 0,C 180,E1 17439.378,E2 17439.378} C_VEL
LIN {X 0,Y 457.027,Z 145.087,A -85,B 0,C 180,E1 17435.82,E2 17435.82} C_VEL
LIN {X 0,Y 457.015,Z 145.12,A -85,B 0,C 180,E1 17432.225,E2 17432.225} C_VEL
LIN {X 0,Y 457.011,Z 145.082,A -85,B 0,C 180,E1 17428.564,E2 17428.564} C_VEL
LIN {X 0,Y 457.042,Z 145.084,A -85,B 0,C 180,E1 17425.028,E2 17425.028} C_VEL
LIN {X 0,Y 457.047,Z 145.362,A -85,B 0,C 180,E1 17422.601,E2 17422.601} C_VEL
LIN {X 0,Y 458.491,Z 148.854,A -85,B 0,C 180,E1 17421.891,E2 17421.891} C_VEL
LIN {X 0,Y 459.671,Z 150.332,A -85,B 0,C 180,E1 17421.53,E2 17421.53} C_VEL
LIN {X 0,Y 461.657,Z 154.307,A -85,B 0,C 180,E1 17420.771,E2 17420.771} C_VEL
LIN {X 0,Y 466.909,Z 164.394,A -85,B 0,C 180,E1 17418.896,E2 17418.896} C_VEL
LIN {X 0,Y 474.58,Z 179.921,A -85,B 0,C 180,E1 17416.271,E2 17416.271} C_VEL
LIN {X 0,Y 482.652,Z 197.818,A -85,B 0,C 180,E1 17413.586,E2 17413.586} C_VEL
LIN {X 0,Y 482.225,Z 205.394,A -85,B 0,C 180,E1 17413.013,E2 17413.013} C_VEL
LIN {X 0,Y 487.362,Z 238.107,A -85,B 0,C 180,E1 17411.757,E2 17411.757} C_VEL
LIN {X 0,Y 484.701,Z 357.497,A -85,B 0,C 180,E1 17409.784,E2 17409.784} C_VEL
LIN {X 0,Y 483.818,Z 365.201,A -85,B 0,C 180,E1 17409.737,E2 17409.737} C_VEL
LIN {X 0,Y 478.776,Z 385.797,A -85,B 0,C 180,E1 17409.906,E2 17409.906} C_VEL
LIN {X 0,Y 478.081,Z 392.408,A -85,B 0,C 180,E1 17409.859,E2 17409.859} C_VEL
LIN {X 0,Y 475.264,Z 515.151,A -85,B 0,C 180,E1 17407.815,E2 17407.815} C_VEL
LIN {X 0,Y 474.032,Z 536.178,A -85,B 0,C 180,E1 17407.274,E2 17407.274} C_VEL
LIN {X 0,Y 472.404,Z 556.976,A -85,B 0,C 180,E1 17406.531,E2 17406.531} C_VEL
LIN {X 0,Y 470.404,Z 576.468,A -85,B 0,C 180,E1 17405.618,E2 17405.618} C_VEL
LIN {X 0,Y 467.952,Z 596.947,A -85,B 0,C 180,E1 17404.419,E2 17404.419} C_VEL
LIN {X 0,Y 465.439,Z 615.896,A -85,B 0,C 180,E1 17403.068,E2 17403.068} C_VEL
LIN {X 0,Y 462.657,Z 634.533,A -85,B 0,C 180,E1 17401.46,E2 17401.46} C_VEL
LIN {X 0,Y 459.953,Z 652.235,A -85,B 0,C 180,E1 17399.657,E2 17399.657} C_VEL
LIN {X 0,Y 457.436,Z 668.53,A -85,B 0,C 180,E1 17397.718,E2 17397.718} C_VEL
LIN {X 0,Y 455.029,Z 684.249,A -85,B 0,C 180,E1 17395.51,E2 17395.51} C_VEL
LIN {X 0,Y 452.937,Z 698.737,A -85,B 0,C 180,E1 17393.137,E2 17393.137} C_VEL
LIN {X 0,Y 451.235,Z 711.792,A -85,B 0,C 180,E1 17390.628,E2 17390.628} C_VEL
LIN {X 0,Y 449.832,Z 724.592,A -85,B 0,C 180,E1 17387.728,E2 17387.728} C_VEL
LIN {X 0,Y 449.011,Z 733.854,A -85,B 0,C 180,E1 17385.234,E2 17385.234} C_VEL
LIN {X 0,Y 448.43,Z 742.198,A -85,B 0,C 180,E1 17382.49,E2 17382.49} C_VEL
LIN {X 0,Y 448.121,Z 748.54,A -85,B 0,C 180,E1 17379.892,E2 17379.892} C_VEL
LIN {X 0,Y 447.977,Z 753.241,A -85,B 0,C 180,E1 17377.309,E2 17377.309} C_VEL
LIN {X 0,Y 447.921,Z 756.79,A -85,B 0,C 180,E1 17374.481,E2 17374.481} C_VEL
LIN {X 0,Y 447.907,Z 758.558,A -85,B 0,C 180,E1 17371.919,E2 17371.919} C_VEL
LIN {X 0,Y 447.905,Z 758.876,A -85,B 0,C 180,E1 17369.233,E2 17369.233} C_VEL
LIN {X 0,Y 447.915,Z 757.778,A -85,B 0,C 180,E1 17366.545,E2 17366.545} C_VEL
LIN {X 0,Y 447.945,Z 755.017,A -85,B 0,C 180,E1 17363.85,E2 17363.85} C_VEL
LIN {X 0,Y 448.049,Z 750.497,A -85,B 0,C 180,E1 17361.013,E2 17361.013} C_VEL
LIN {X 0,Y 448.314,Z 744.548,A -85,B 0,C 180,E1 17358.291,E2 17358.291} C_VEL
LIN {X 0,Y 448.762,Z 737.116,A -85,B 0,C 180,E1 17355.682,E2 17355.682} C_VEL
LIN {X 0,Y 449.54,Z 727.516,A -85,B 0,C 180,E1 17352.927,E2 17352.927} C_VEL
LIN {X 0,Y 450.672,Z 716.515,A -85,B 0,C 180,E1 17350.293,E2 17350.293} C_VEL
LIN {X 0,Y 452.191,Z 704.273,A -85,B 0,C 180,E1 17347.784,E2 17347.784} C_VEL
LIN {X 0,Y 454.075,Z 690.667,A -85,B 0,C 180,E1 17345.408,E2 17345.408} C_VEL
LIN {X 0,Y 456.309,Z 675.772,A -85,B 0,C 180,E1 17343.168,E2 17343.168} C_VEL
LIN {X 0,Y 458.796,Z 659.747,A -85,B 0,C 180,E1 17341.108,E2 17341.108} C_VEL
LIN {X 0,Y 461.423,Z 642.686,A -85,B 0,C 180,E1 17339.245,E2 17339.245} C_VEL
LIN {X 0,Y 464.249,Z 623.863,A -85,B 0,C 180,E1 17337.498,E2 17337.498} C_VEL
LIN {X 0,Y 466.95,Z 604.898,A -85,B 0,C 180,E1 17336.024,E2 17336.024} C_VEL
LIN {X 0,Y 469.33,Z 585.892,A -85,B 0,C 180,E1 17334.812,E2 17334.812} C_VEL
LIN {X 0,Y 471.536,Z 565.887,A -85,B 0,C 180,E1 17333.768,E2 17333.768} C_VEL
LIN {X 0,Y 473.364,Z 545.319,A -85,B 0,C 180,E1 17332.932,E2 17332.932} C_VEL
LIN {X 0,Y 474.788,Z 524.311,A -85,B 0,C 180,E1 17332.308,E2 17332.308} C_VEL
LIN {X 0,Y 475.716,Z 502.209,A -85,B 0,C 180,E1 17331.858,E2 17331.858} C_VEL
LIN {X 0,Y 480.714,Z 276.255,A -85,B 0,C 180,E1 17328.124,E2 17328.124} C_VEL
LIN {X 0,Y 481.525,Z 238.198,A -85,B 0,C 180,E1 17327.466,E2 17327.466} C_VEL
LIN {X 0,Y 476.163,Z 203.61,A -85,B 0,C 180,E1 17326.075,E2 17326.075} C_VEL
LIN {X 0,Y 476.245,Z 201.496,A -85,B 0,C 180,E1 17325.891,E2 17325.891} C_VEL
LIN {X 0,Y 468.111,Z 183.497,A -85,B 0,C 180,E1 17323.118,E2 17323.118} C_VEL
LIN {X 0,Y 460.964,Z 168.921,A -85,B 0,C 180,E1 17320.596,E2 17320.596} C_VEL
LIN {X 0,Y 455.716,Z 159.129,A -85,B 0,C 180,E1 17318.704,E2 17318.704} C_VEL
LIN {X 0,Y 453.718,Z 155.299,A -85,B 0,C 180,E1 17317.94,E2 17317.94} C_VEL
LIN {X 0,Y 451.789,Z 151.503,A -85,B 0,C 180,E1 17317.17,E2 17317.17} C_VEL
LIN {X 0,Y 449.417,Z 147.582,A -85,B 0,C 180,E1 17316.285,E2 17316.285} C_VEL
LIN {X 0,Y 449.065,Z 146.128,A -85,B 0,C 180,E1 17315.897,E2 17315.897} C_VEL
LIN {X 0,Y 449.08,Z 146.081,A -85,B 0,C 180,E1 17312.217,E2 17312.217} C_VEL
LIN {X 0,Y 449.122,Z 146.099,A -85,B 0,C 180,E1 17308.597,E2 17308.597} C_VEL
LIN {X 0,Y 449.11,Z 146.059,A -85,B 0,C 180,E1 17304.884,E2 17304.884} C_VEL
LIN {X 0,Y 449.087,Z 146.092,A -85,B 0,C 180,E1 17301.279,E2 17301.279} C_VEL
LIN {X 0,Y 449.077,Z 146.08,A -85,B 0,C 180,E1 17297.626,E2 17297.626} C_VEL
LIN {X 0,Y 449.085,Z 146.097,A -85,B 0,C 180,E1 17293.904,E2 17293.904} C_VEL
LIN {X 0,Y 449.104,Z 146.098,A -85,B 0,C 180,E1 17290.259,E2 17290.259} C_VEL
LIN {X 0,Y 449.138,Z 146.094,A -85,B 0,C 180,E1 17286.648,E2 17286.648} C_VEL
LIN {X 0,Y 449.126,Z 146.095,A -85,B 0,C 180,E1 17282.935,E2 17282.935} C_VEL
LIN {X 0,Y 449.104,Z 146.097,A -85,B 0,C 180,E1 17279.362,E2 17279.362} C_VEL
LIN {X 0,Y 449.098,Z 146.1,A -85,B 0,C 180,E1 17275.659,E2 17275.659} C_VEL
LIN {X 0,Y 449.104,Z 146.101,A -85,B 0,C 180,E1 17271.937,E2 17271.937} C_VEL
LIN {X 0,Y 449.124,Z 146.101,A -85,B 0,C 180,E1 17268.312,E2 17268.312} C_VEL
LIN {X 0,Y 449.133,Z 146.05,A -85,B 0,C 180,E1 17264.561,E2 17264.561} C_VEL
LIN {X 0,Y 449.138,Z 146.095,A -85,B 0,C 180,E1 17260.763,E2 17260.763} C_VEL
LIN {X 0,Y 449.136,Z 146.071,A -85,B 0,C 180,E1 17256.933,E2 17256.933} C_VEL
LIN {X 0,Y 449.124,Z 146.061,A -85,B 0,C 180,E1 17253.214,E2 17253.214} C_VEL
LIN {X 0,Y 449.123,Z 146.091,A -85,B 0,C 180,E1 17249.489,E2 17249.489} C_VEL
LIN {X 0,Y 449.154,Z 146.262,A -85,B 0,C 180,E1 17246.338,E2 17246.338} C_VEL
LIN {X 0,Y 449.682,Z 148.192,A -85,B 0,C 180,E1 17245.923,E2 17245.923} C_VEL
LIN {X 0,Y 451.905,Z 151.423,A -85,B 0,C 180,E1 17245.168,E2 17245.168} C_VEL
LIN {X 0,Y 453.79,Z 155.208,A -85,B 0,C 180,E1 17244.431,E2 17244.431} C_VEL
LIN {X 0,Y 455.112,Z 157.673,A -85,B 0,C 180,E1 17243.945,E2 17243.945} C_VEL
LIN {X 0,Y 457.939,Z 162.85,A -85,B 0,C 180,E1 17242.943,E2 17242.943} C_VEL
LIN {X 0,Y 461.385,Z 168.932,A -85,B 0,C 180,E1 17241.858,E2 17241.858} C_VEL
LIN {X 0,Y 472.715,Z 184.774,A -85,B 0,C 180,E1 17239.925,E2 17239.925} C_VEL
LIN {X 0,Y 485.699,Z 204.442,A -85,B 0,C 180,E1 17237.868,E2 17237.868} C_VEL
LIN {X 0,Y 486.172,Z 205.773,A -85,B 0,C 180,E1 17237.783,E2 17237.783} C_VEL
LIN {X 0,Y 480.187,Z 417.423,A -85,B 0,C 180,E1 17234.037,E2 17234.037} C_VEL
LIN {X 0,Y 477.634,Z 512.615,A -85,B 0,C 180,E1 17232.366,E2 17232.366} C_VEL
LIN {X 0,Y 476.277,Z 535.497,A -85,B 0,C 180,E1 17231.768,E2 17231.768} C_VEL
LIN {X 0,Y 474.599,Z 558.108,A -85,B 0,C 180,E1 17230.977,E2 17230.977} C_VEL
LIN {X 0,Y 472.629,Z 579.352,A -85,B 0,C 180,E1 17230.02,E2 17230.02} C_VEL
LIN {X 0,Y 470.212,Z 602.196,A -85,B 0,C 180,E1 17228.757,E2 17228.757} C_VEL
LIN {X 0,Y 467.908,Z 621.951,A -85,B 0,C 180,E1 17227.439,E2 17227.439} C_VEL
LIN {X 0,Y 465.308,Z 642.153,A -85,B 0,C 180,E1 17225.841,E2 17225.841} C_VEL
LIN {X 0,Y 462.737,Z 660.924,A -85,B 0,C 180,E1 17224.112,E2 17224.112} C_VEL
LIN {X 0,Y 460.175,Z 679.001,A -85,B 0,C 180,E1 17222.162,E2 17222.162} C_VEL
LIN {X 0,Y 457.85,Z 695.42,A -85,B 0,C 180,E1 17220.142,E2 17220.142} C_VEL
LIN {X 0,Y 455.799,Z 709.316,A -85,B 0,C 180,E1 17218.135,E2 17218.135} C_VEL
LIN {X 0,Y 453.704,Z 723.734,A -85,B 0,C 180,E1 17215.73,E2 17215.73} C_VEL
LIN {X 0,Y 451.938,Z 736.808,A -85,B 0,C 180,E1 17213.191,E2 17213.191} C_VEL
LIN {X 0,Y 450.525,Z 748.752,A -85,B 0,C 180,E1 17210.52,E2 17210.52} C_VEL
LIN {X 0,Y 449.443,Z 759.145,A -85,B 0,C 180,E1 17207.744,E2 17207.744} C_VEL
LIN {X 0,Y 448.706,Z 768.286,A -85,B 0,C 180,E1 17204.848,E2 17204.848} C_VEL
LIN {X 0,Y 448.293,Z 774.956,A -85,B 0,C 180,E1 17202.232,E2 17202.232} C_VEL
LIN {X 0,Y 448.049,Z 780.809,A -85,B 0,C 180,E1 17199.375,E2 17199.375} C_VEL
LIN {X 0,Y 447.949,Z 784.819,A -85,B 0,C 180,E1 17196.65,E2 17196.65} C_VEL
LIN {X 0,Y 447.913,Z 787.67,A -85,B 0,C 180,E1 17193.787,E2 17193.787} C_VEL
LIN {X 0,Y 447.912,Z 788.826,A -85,B 0,C 180,E1 17191.023,E2 17191.023} C_VEL
LIN {X 0,Y 447.901,Z 788.713,A -85,B 0,C 180,E1 17188.337,E2 17188.337} C_VEL
LIN {X 0,Y 447.905,Z 787.068,A -85,B 0,C 180,E1 17185.519,E2 17185.519} C_VEL
LIN {X 0,Y 447.96,Z 784.32,A -85,B 0,C 180,E1 17182.949,E2 17182.949} C_VEL
LIN {X 0,Y 448.078,Z 779.591,A -85,B 0,C 180,E1 17179.977,E2 17179.977} C_VEL
LIN {X 0,Y 448.34,Z 774.045,A -85,B 0,C 180,E1 17177.376,E2 17177.376} C_VEL
LIN {X 0,Y 448.868,Z 765.958,A -85,B 0,C 180,E1 17174.364,E2 17174.364} C_VEL
LIN {X 0,Y 449.623,Z 757.296,A -85,B 0,C 180,E1 17171.722,E2 17171.722} C_VEL
LIN {X 0,Y 450.832,Z 745.866,A -85,B 0,C 180,E1 17168.808,E2 17168.808} C_VEL
LIN {X 0,Y 452.368,Z 733.627,A -85,B 0,C 180,E1 17166.142,E2 17166.142} C_VEL
LIN {X 0,Y 454.238,Z 719.882,A -85,B 0,C 180,E1 17163.601,E2 17163.601} C_VEL
LIN {X 0,Y 456.478,Z 704.885,A -85,B 0,C 180,E1 17161.181,E2 17161.181} C_VEL
LIN {X 0,Y 458.664,Z 689.567,A -85,B 0,C 180,E1 17159.112,E2 17159.112} C_VEL
LIN {X 0,Y 461.28,Z 671.255,A -85,B 0,C 180,E1 17156.967,E2 17156.967} C_VEL
LIN {X 0,Y 463.676,Z 654.189,A -85,B 0,C 180,E1 17155.243,E2 17155.243} C_VEL
LIN {X 0,Y 466.453,Z 633.292,A -85,B 0,C 180,E1 17153.424,E2 17153.424} C_VEL
LIN {X 0,Y 468.785,Z 614.661,A -85,B 0,C 180,E1 17152.048,E2 17152.048} C_VEL
LIN {X 0,Y 471.223,Z 593.122,A -85,B 0,C 180,E1 17150.712,E2 17150.712} C_VEL
LIN {X 0,Y 473.293,Z 572.715,A -85,B 0,C 180,E1 17149.656,E2 17149.656} C_VEL
LIN {X 0,Y 475.207,Z 549.855,A -85,B 0,C 180,E1 17148.711,E2 17148.711} C_VEL
LIN {X 0,Y 476.85,Z 526.804,A -85,B 0,C 180,E1 17147.975,E2 17147.975} C_VEL
LIN {X 0,Y 477.961,Z 503.979,A -85,B 0,C 180,E1 17147.468,E2 17147.468} C_VEL
LIN {X 0,Y 483.582,Z 295.461,A -85,B 0,C 180,E1 17143.81,E2 17143.81} C_VEL
LIN {X 0,Y 486.085,Z 205.072,A -85,B 0,C 180,E1 17142.19,E2 17142.19} C_VEL
LIN {X 0,Y 473.816,Z 186.457,A -85,B 0,C 180,E1 17140.26,E2 17140.26} C_VEL
LIN {X 0,Y 464.388,Z 173.078,A -85,B 0,C 180,E1 17138.677,E2 17138.677} C_VEL
LIN {X 0,Y 460.417,Z 167.473,A -85,B 0,C 180,E1 17137.921,E2 17137.921} C_VEL
LIN {X 0,Y 456.175,Z 159.573,A -85,B 0,C 180,E1 17136.44,E2 17136.44} C_VEL
LIN {X 0,Y 453.763,Z 155.176,A -85,B 0,C 180,E1 17135.571,E2 17135.571} C_VEL
LIN {X 0,Y 451.442,Z 150.805,A -85,B 0,C 180,E1 17134.695,E2 17134.695} C_VEL
LIN {X 0,Y 449.658,Z 148.135,A -85,B 0,C 180,E1 17134.079,E2 17134.079} C_VEL
LIN {X 0,Y 449.154,Z 146.258,A -85,B 0,C 180,E1 17133.662,E2 17133.662} C_VEL
LIN {X 0,Y 449.123,Z 146.106,A -85,B 0,C 180,E1 17130.005,E2 17130.005} C_VEL
LIN {X 0,Y 449.113,Z 146.07,A -85,B 0,C 180,E1 17126.211,E2 17126.211} C_VEL
LIN {X 0,Y 449.112,Z 146.063,A -85,B 0,C 180,E1 17122.499,E2 17122.499} C_VEL
LIN {X 0,Y 449.13,Z 146.102,A -85,B 0,C 180,E1 17118.832,E2 17118.832} C_VEL
LIN {X 0,Y 449.134,Z 146.05,A -85,B 0,C 180,E1 17115.097,E2 17115.097} C_VEL
LIN {X 0,Y 449.136,Z 146.095,A -85,B 0,C 180,E1 17111.297,E2 17111.297} C_VEL
LIN {X 0,Y 449.137,Z 146.093,A -85,B 0,C 180,E1 17107.547,E2 17107.547} C_VEL
LIN {X 0,Y 449.112,Z 146.095,A -85,B 0,C 180,E1 17103.829,E2 17103.829} C_VEL
LIN {X 0,Y 449.096,Z 146.095,A -85,B 0,C 180,E1 17100.255,E2 17100.255} C_VEL
LIN {X 0,Y 449.099,Z 146.093,A -85,B 0,C 180,E1 17096.554,E2 17096.554} C_VEL
LIN {X 0,Y 449.124,Z 146.092,A -85,B 0,C 180,E1 17092.967,E2 17092.967} C_VEL
LIN {X 0,Y 449.132,Z 146.091,A -85,B 0,C 180,E1 17089.222,E2 17089.222} C_VEL
LIN {X 0,Y 449.117,Z 146.092,A -85,B 0,C 180,E1 17085.558,E2 17085.558} C_VEL
LIN {X 0,Y 449.087,Z 146.07,A -85,B 0,C 180,E1 17081.926,E2 17081.926} C_VEL
LIN {X 0,Y 449.08,Z 146.103,A -85,B 0,C 180,E1 17078.309,E2 17078.309} C_VEL
LIN {X 0,Y 449.085,Z 146.061,A -85,B 0,C 180,E1 17074.676,E2 17074.676} C_VEL
LIN {X 0,Y 449.114,Z 146.094,A -85,B 0,C 180,E1 17071.034,E2 17071.034} C_VEL
LIN {X 0,Y 449.121,Z 146.086,A -85,B 0,C 180,E1 17067.299,E2 17067.299} C_VEL
LIN {X 0,Y 449.101,Z 146.298,A -85,B 0,C 180,E1 17063.915,E2 17063.915} C_VEL
LIN {X 0,Y 450.121,Z 149.077,A -85,B 0,C 180,E1 17063.306,E2 17063.306} C_VEL
LIN {X 0,Y 451.874,Z 151.789,A -85,B 0,C 180,E1 17062.679,E2 17062.679} C_VEL
LIN {X 0,Y 453.866,Z 155.464,A -85,B 0,C 180,E1 17061.914,E2 17061.914} C_VEL
LIN {X 0,Y 459.653,Z 166.576,A -85,B 0,C 180,E1 17059.755,E2 17059.755} C_VEL
LIN {X 0,Y 465.731,Z 178.633,A -85,B 0,C 180,E1 17057.604,E2 17057.604} C_VEL
LIN {X 0,Y 473.882,Z 196.178,A -85,B 0,C 180,E1 17054.805,E2 17054.805} C_VEL
LIN {X 0,Y 476.317,Z 201.687,A -85,B 0,C 180,E1 17053.99,E2 17053.99} C_VEL
LIN {X 0,Y 476.279,Z 205.142,A -85,B 0,C 180,E1 17053.756,E2 17053.756} C_VEL
LIN {X 0,Y 481.623,Z 239.661,A -85,B 0,C 180,E1 17052.399,E2 17052.399} C_VEL
LIN {X 0,Y 478.081,Z 392.408,A -85,B 0,C 180,E1 17049.859,E2 17049.859} C_VEL
LIN {X 0,Y 477.186,Z 400.113,A -85,B 0,C 180,E1 17049.812,E2 17049.812} C_VEL
LIN {X 0,Y 472.141,Z 420.707,A -85,B 0,C 180,E1 17049.986,E2 17049.986} C_VEL
LIN {X 0,Y 471.437,Z 427.319,A -85,B 0,C 180,E1 17049.939,E2 17049.939} C_VEL
LIN {X 0,Y 469.257,Z 516.229,A -85,B 0,C 180,E1 17048.444,E2 17048.444} C_VEL
LIN {X 0,Y 467.958,Z 537.27,A -85,B 0,C 180,E1 17047.894,E2 17047.894} C_VEL
LIN {X 0,Y 466.236,Z 558.266,A -85,B 0,C 180,E1 17047.133,E2 17047.133} C_VEL
LIN {X 0,Y 464.234,Z 577.175,A -85,B 0,C 180,E1 17046.242,E2 17046.242} C_VEL
LIN {X 0,Y 461.632,Z 597.736,A -85,B 0,C 180,E1 17045.026,E2 17045.026} C_VEL
LIN {X 0,Y 459.012,Z 616.336,A -85,B 0,C 180,E1 17043.684,E2 17043.684} C_VEL
LIN {X 0,Y 456.137,Z 634.409,A -85,B 0,C 180,E1 17042.11,E2 17042.11} C_VEL
LIN {X 0,Y 453.091,Z 652.83,A -85,B 0,C 180,E1 17040.207,E2 17040.207} C_VEL
LIN {X 0,Y 450.29,Z 669.57,A -85,B 0,C 180,E1 17038.172,E2 17038.172} C_VEL
LIN {X 0,Y 447.738,Z 685.045,A -85,B 0,C 180,E1 17035.956,E2 17035.956} C_VEL
LIN {X 0,Y 445.462,Z 699.367,A -85,B 0,C 180,E1 17033.548,E2 17033.548} C_VEL
LIN {X 0,Y 443.524,Z 712.955,A -85,B 0,C 180,E1 17030.866,E2 17030.866} C_VEL
LIN {X 0,Y 442.105,Z 724.412,A -85,B 0,C 180,E1 17028.185,E2 17028.185} C_VEL
LIN {X 0,Y 441.119,Z 733.889,A -85,B 0,C 180,E1 17025.513,E2 17025.513} C_VEL
LIN {X 0,Y 440.486,Z 742.2,A -85,B 0,C 180,E1 17022.719,E2 17022.719} C_VEL
LIN {X 0,Y 440.144,Z 748.542,A -85,B 0,C 180,E1 17020.074,E2 17020.074} C_VEL
LIN {X 0,Y 439.98,Z 753.242,A -85,B 0,C 180,E1 17017.442,E2 17017.442} C_VEL
LIN {X 0,Y 439.921,Z 756.79,A -85,B 0,C 180,E1 17014.562,E2 17014.562} C_VEL
LIN {X 0,Y 439.907,Z 758.558,A -85,B 0,C 180,E1 17011.954,E2 17011.954} C_VEL
LIN {X 0,Y 439.905,Z 758.876,A -85,B 0,C 180,E1 17009.219,E2 17009.219} C_VEL
LIN {X 0,Y 439.915,Z 757.777,A -85,B 0,C 180,E1 17006.482,E2 17006.482} C_VEL
LIN {X 0,Y 439.947,Z 755.016,A -85,B 0,C 180,E1 17003.737,E2 17003.737} C_VEL
LIN {X 0,Y 440.069,Z 750.495,A -85,B 0,C 180,E1 17000.849,E2 17000.849} C_VEL
LIN {X 0,Y 440.355,Z 744.546,A -85,B 0,C 180,E1 16998.076,E2 16998.076} C_VEL
LIN {X 0,Y 440.846,Z 737.113,A -85,B 0,C 180,E1 16995.419,E2 16995.419} C_VEL
LIN {X 0,Y 441.777,Z 727.234,A -85,B 0,C 180,E1 16992.482,E2 16992.482} C_VEL
LIN {X 0,Y 443.047,Z 716.662,A -85,B 0,C 180,E1 16989.855,E2 16989.855} C_VEL
LIN {X 0,Y 444.754,Z 704.173,A -85,B 0,C 180,E1 16987.253,E2 16987.253} C_VEL
LIN {X 0,Y 446.828,Z 690.558,A -85,B 0,C 180,E1 16984.84,E2 16984.84} C_VEL
LIN {X 0,Y 449.343,Z 675.208,A -85,B 0,C 180,E1 16982.51,E2 16982.51} C_VEL
LIN {X 0,Y 452.024,Z 659.304,A -85,B 0,C 180,E1 16980.445,E2 16980.445} C_VEL
LIN {X 0,Y 454.812,Z 642.547,A -85,B 0,C 180,E1 16978.6,E2 16978.6} C_VEL
LIN {X 0,Y 457.838,Z 623.687,A -85,B 0,C 180,E1 16976.836,E2 16976.836} C_VEL
LIN {X 0,Y 460.729,Z 604.655,A -85,B 0,C 180,E1 16975.35,E2 16975.35} C_VEL
LIN {X 0,Y 463.242,Z 585.485,A -85,B 0,C 180,E1 16974.127,E2 16974.127} C_VEL
LIN {X 0,Y 465.614,Z 564.337,A -85,B 0,C 180,E1 16973.04,E2 16973.04} C_VEL
LIN {X 0,Y 467.539,Z 543.482,A -85,B 0,C 180,E1 16972.212,E2 16972.212} C_VEL
LIN {X 0,Y 468.898,Z 522.751,A -85,B 0,C 180,E1 16971.618,E2 16971.618} C_VEL
LIN {X 0,Y 469.872,Z 496.935,A -85,B 0,C 180,E1 16971.12,E2 16971.12} C_VEL
LIN {X 0,Y 475.225,Z 268.468,A -85,B 0,C 180,E1 16967.314,E2 16967.314} C_VEL
LIN {X 0,Y 475.83,Z 239.593,A -85,B 0,C 180,E1 16966.802,E2 16966.802} C_VEL
LIN {X 0,Y 470.47,Z 205.797,A -85,B 0,C 180,E1 16965.416,E2 16965.416} C_VEL
LIN {X 0,Y 468.759,Z 202.834,A -85,B 0,C 180,E1 16965.085,E2 16965.085} C_VEL
LIN {X 0,Y 461.126,Z 186.039,A -85,B 0,C 180,E1 16962.403,E2 16962.403} C_VEL
LIN {X 0,Y 455.133,Z 173.844,A -85,B 0,C 180,E1 16960.231,E2 16960.231} C_VEL
LIN {X 0,Y 448.706,Z 161.424,A -85,B 0,C 180,E1 16957.792,E2 16957.792} C_VEL
LIN {X 0,Y 445.711,Z 156.083,A -85,B 0,C 180,E1 16956.635,E2 16956.635} C_VEL
LIN {X 0,Y 443.535,Z 151.867,A -85,B 0,C 180,E1 16955.723,E2 16955.723} C_VEL
LIN {X 0,Y 441.529,Z 148.666,A -85,B 0,C 180,E1 16954.941,E2 16954.941} C_VEL
LIN {X 0,Y 441.171,Z 147.133,A -85,B 0,C 180,E1 16954.526,E2 16954.526} C_VEL
LIN {X 0,Y 441.176,Z 147.047,A -85,B 0,C 180,E1 16950.804,E2 16950.804} C_VEL
LIN {X 0,Y 441.143,Z 147.079,A -85,B 0,C 180,E1 16947.248,E2 16947.248} C_VEL
LIN {X 0,Y 441.132,Z 147.072,A -85,B 0,C 180,E1 16943.652,E2 16943.652} C_VEL
LIN {X 0,Y 441.135,Z 147.049,A -85,B 0,C 180,E1 16939.876,E2 16939.876} C_VEL
LIN {X 0,Y 441.157,Z 147.096,A -85,B 0,C 180,E1 16936.187,E2 16936.187} C_VEL
LIN {X 0,Y 441.188,Z 147.093,A -85,B 0,C 180,E1 16932.566,E2 16932.566} C_VEL
LIN {X 0,Y 441.197,Z 147.089,A -85,B 0,C 180,E1 16928.734,E2 16928.734} C_VEL
LIN {X 0,Y 441.179,Z 147.091,A -85,B 0,C 180,E1 16925.071,E2 16925.071} C_VEL
LIN {X 0,Y 441.161,Z 147.093,A -85,B 0,C 180,E1 16921.429,E2 16921.429} C_VEL
LIN {X 0,Y 441.158,Z 147.092,A -85,B 0,C 180,E1 16917.662,E2 16917.662} C_VEL
LIN {X 0,Y 441.161,Z 147.087,A -85,B 0,C 180,E1 16913.885,E2 16913.885} C_VEL
LIN {X 0,Y 441.178,Z 147.081,A -85,B 0,C 180,E1 16910.214,E2 16910.214} C_VEL
LIN {X 0,Y 441.194,Z 147.063,A -85,B 0,C 180,E1 16906.457,E2 16906.457} C_VEL
LIN {X 0,Y 441.196,Z 147.067,A -85,B 0,C 180,E1 16902.73,E2 16902.73} C_VEL
LIN {X 0,Y 441.191,Z 147.043,A -85,B 0,C 180,E1 16899.015,E2 16899.015} C_VEL
LIN {X 0,Y 441.189,Z 147.091,A -85,B 0,C 180,E1 16895.212,E2 16895.212} C_VEL
LIN {X 0,Y 441.181,Z 147.059,A -85,B 0,C 180,E1 16891.433,E2 16891.433} C_VEL
LIN {X 0,Y 441.204,Z 147.258,A -85,B 0,C 180,E1 16887.733,E2 16887.733} C_VEL
LIN {X 0,Y 441.814,Z 149.307,A -85,B 0,C 180,E1 16887.257,E2 16887.257} C_VEL
LIN {X 0,Y 444.193,Z 152.966,A -85,B 0,C 180,E1 16886.377,E2 16886.377} C_VEL
LIN {X 0,Y 446.132,Z 156.544,A -85,B 0,C 180,E1 16885.614,E2 16885.614} C_VEL
LIN {X 0,Y 449.839,Z 163.284,A -85,B 0,C 180,E1 16884.22,E2 16884.22} C_VEL
LIN {X 0,Y 453.147,Z 169.267,A -85,B 0,C 180,E1 16883.079,E2 16883.079} C_VEL
LIN {X 0,Y 463.105,Z 182.929,A -85,B 0,C 180,E1 16881.276,E2 16881.276} C_VEL
LIN {X 0,Y 474.522,Z 199.571,A -85,B 0,C 180,E1 16879.357,E2 16879.357} C_VEL
LIN {X 0,Y 480.446,Z 209.112,A -85,B 0,C 180,E1 16878.403,E2 16878.403} C_VEL
LIN {X 0,Y 474.044,Z 421.157,A -85,B 0,C 180,E1 16874.605,E2 16874.605} C_VEL
LIN {X 0,Y 471.322,Z 512.271,A -85,B 0,C 180,E1 16872.969,E2 16872.969} C_VEL
LIN {X 0,Y 469.859,Z 535.326,A -85,B 0,C 180,E1 16872.358,E2 16872.358} C_VEL
LIN {X 0,Y 468.064,Z 558.152,A -85,B 0,C 180,E1 16871.549,E2 16871.549} C_VEL
LIN {X 0,Y 466.092,Z 578.421,A -85,B 0,C 180,E1 16870.627,E2 16870.627} C_VEL
LIN {X 0,Y 463.685,Z 600.163,A -85,B 0,C 180,E1 16869.43,E2 16869.43} C_VEL
LIN {X 0,Y 461.22,Z 620.085,A -85,B 0,C 180,E1 16868.101,E2 16868.101} C_VEL
LIN {X 0,Y 458.352,Z 641.689,A -85,B 0,C 180,E1 16866.394,E2 16866.394} C_VEL
LIN {X 0,Y 455.836,Z 659.263,A -85,B 0,C 180,E1 16864.77,E2 16864.77} C_VEL
LIN {X 0,Y 453.016,Z 678.11,A -85,B 0,C 180,E1 16862.733,E2 16862.733} C_VEL
LIN {X 0,Y 450.476,Z 695.072,A -85,B 0,C 180,E1 16860.622,E2 16860.622} C_VEL
LIN {X 0,Y 448.126,Z 710.566,A -85,B 0,C 180,E1 16858.374,E2 16858.374} C_VEL
LIN {X 0,Y 446.208,Z 723.732,A -85,B 0,C 180,E1 16856.195,E2 16856.195} C_VEL
LIN {X 0,Y 444.299,Z 736.806,A -85,B 0,C 180,E1 16853.613,E2 16853.613} C_VEL
LIN {X 0,Y 442.768,Z 748.725,A -85,B 0,C 180,E1 16850.903,E2 16850.903} C_VEL
LIN {X 0,Y 441.59,Z 759.143,A -85,B 0,C 180,E1 16848.071,E2 16848.071} C_VEL
LIN {X 0,Y 440.786,Z 768.286,A -85,B 0,C 180,E1 16845.121,E2 16845.121} C_VEL
LIN {X 0,Y 440.332,Z 774.955,A -85,B 0,C 180,E1 16842.457,E2 16842.457} C_VEL
LIN {X 0,Y 440.06,Z 780.81,A -85,B 0,C 180,E1 16839.547,E2 16839.547} C_VEL
LIN {X 0,Y 439.955,Z 784.8,A -85,B 0,C 180,E1 16836.787,E2 16836.787} C_VEL
LIN {X 0,Y 439.913,Z 787.632,A -85,B 0,C 180,E1 16833.91,E2 16833.91} C_VEL
LIN {X 0,Y 439.912,Z 788.826,A -85,B 0,C 180,E1 16831.042,E2 16831.042} C_VEL
LIN {X 0,Y 439.901,Z 788.712,A -85,B 0,C 180,E1 16828.307,E2 16828.307} C_VEL
LIN {X 0,Y 439.905,Z 787.068,A -85,B 0,C 180,E1 16825.437,E2 16825.437} C_VEL
LIN {X 0,Y 439.966,Z 784.32,A -85,B 0,C 180,E1 16822.82,E2 16822.82} C_VEL
LIN {X 0,Y 440.101,Z 779.591,A -85,B 0,C 180,E1 16819.793,E2 16819.793} C_VEL
LIN {X 0,Y 440.382,Z 774.045,A -85,B 0,C 180,E1 16817.144,E2 16817.144} C_VEL
LIN {X 0,Y 440.979,Z 765.785,A -85,B 0,C 180,E1 16814.02,E2 16814.02} C_VEL
LIN {X 0,Y 441.793,Z 757.312,A -85,B 0,C 180,E1 16811.392,E2 16811.392} C_VEL
LIN {X 0,Y 443.108,Z 745.865,A -85,B 0,C 180,E1 16808.42,E2 16808.42} C_VEL
LIN {X 0,Y 444.767,Z 733.629,A -85,B 0,C 180,E1 16805.708,E2 16805.708} C_VEL
LIN {X 0,Y 446.66,Z 720.62,A -85,B 0,C 180,E1 16803.261,E2 16803.261} C_VEL
LIN {X 0,Y 448.938,Z 705.278,A -85,B 0,C 180,E1 16800.814,E2 16800.814} C_VEL
LIN {X 0,Y 451.326,Z 689.273,A -85,B 0,C 180,E1 16798.628,E2 16798.628} C_VEL
LIN {X 0,Y 454.11,Z 670.936,A -85,B 0,C 180,E1 16796.452,E2 16796.452} C_VEL
LIN {X 0,Y 456.655,Z 653.679,A -85,B 0,C 180,E1 16794.689,E2 16794.689} C_VEL
LIN {X 0,Y 459.554,Z 632.731,A -85,B 0,C 180,E1 16792.861,E2 16792.861} C_VEL
LIN {X 0,Y 462.317,Z 611.853,A -85,B 0,C 180,E1 16791.317,E2 16791.317} C_VEL
LIN {X 0,Y 464.728,Z 591.063,A -85,B 0,C 180,E1 16790.044,E2 16790.044} C_VEL
LIN {X 0,Y 467.035,Z 568.917,A -85,B 0,C 180,E1 16788.911,E2 16788.911} C_VEL
LIN {X 0,Y 468.987,Z 546.76,A -85,B 0,C 180,E1 16788.019,E2 16788.019} C_VEL
LIN {X 0,Y 470.73,Z 522.526,A -85,B 0,C 180,E1 16787.281,E2 16787.281} C_VEL
LIN {X 0,Y 471.84,Z 499.747,A -85,B 0,C 180,E1 16786.785,E2 16786.785} C_VEL
LIN {X 0,Y 478.033,Z 287.837,A -85,B 0,C 180,E1 16783.011,E2 16783.011} C_VEL
LIN {X 0,Y 480.315,Z 208.598,A -85,B 0,C 180,E1 16781.57,E2 16781.57} C_VEL
LIN {X 0,Y 467.621,Z 189.323,A -85,B 0,C 180,E1 16779.502,E2 16779.502} C_VEL
LIN {X 0,Y 456.909,Z 174.336,A -85,B 0,C 180,E1 16777.628,E2 16777.628} C_VEL
LIN {X 0,Y 452.57,Z 168.337,A -85,B 0,C 180,E1 16776.778,E2 16776.778} C_VEL
LIN {X 0,Y 448.655,Z 161.096,A -85,B 0,C 180,E1 16775.35,E2 16775.35} C_VEL
LIN {X 0,Y 446.1,Z 156.506,A -85,B 0,C 180,E1 16774.389,E2 16774.389} C_VEL
LIN {X 0,Y 444.113,Z 152.725,A -85,B 0,C 180,E1 16773.594,E2 16773.594} C_VEL
LIN {X 0,Y 441.505,Z 148.501,A -85,B 0,C 180,E1 16772.602,E2 16772.602} C_VEL
LIN {X 0,Y 441.186,Z 147.125,A -85,B 0,C 180,E1 16772.203,E2 16772.203} C_VEL
LIN {X 0,Y 441.18,Z 147.057,A -85,B 0,C 180,E1 16768.42,E2 16768.42} C_VEL
LIN {X 0,Y 441.186,Z 147.094,A -85,B 0,C 180,E1 16764.645,E2 16764.645} C_VEL
LIN {X 0,Y 441.192,Z 147.043,A -85,B 0,C 180,E1 16760.981,E2 16760.981} C_VEL
LIN {X 0,Y 441.195,Z 147.068,A -85,B 0,C 180,E1 16757.27,E2 16757.27} C_VEL
LIN {X 0,Y 441.196,Z 147.063,A -85,B 0,C 180,E1 16753.498,E2 16753.498} C_VEL
LIN {X 0,Y 441.18,Z 147.08,A -85,B 0,C 180,E1 16749.786,E2 16749.786} C_VEL
LIN {X 0,Y 441.164,Z 147.087,A -85,B 0,C 180,E1 16746.115,E2 16746.115} C_VEL
